# B&R Automation Studio project NAINV104C00R8L515F00 (part 2)

### Update LogProgram.txt
```
2023_08-10(R8)
Add LCSLF Phase2

Add Display of the Languages and Time
	UI	- Act_Background - P1000_ LangTime - Update the arrangement and display of the Languages and time
	NtParam - Add Chinese & German Prep

Manual Accept Condition Modification
	1)	LFFollower, Follower1, Follower2, etc.:
 		> Act_Background_AccData Script
	2) LCSLF:
	    > Act_Main Script
	3) USHermes:
    	> Act_Background_AccData Script
	UI:
	4) Act_OptP0200ToP0201AccDat

After power cycle the machine, buzzer will sound on due to the safety relay haven’t reset.

	DInput > Act_Background

Debug for Inshutter Hide in UI when Inlet Shutter disable in Ntparam.

2023-07-03(R7)
Add - Invert Once(PassThrough > Return & Invert) and Invert Twice(Invert > Return & Invert) Mode with Clmap(NoStopper)

	UI		> P0200 - add Upstream 2 Indication,PCB Reset
			> P1023 - add Upstream Selection
			> P0940	- Communication Control

	SMEMA	> Add - USSMEMA 2

	Conv	> Add - Conveyor Direction Access in Act_Link

	Operations	> Add - Act_OpsClampNoStopperInvOnceAndTwice, Act_Link

	McParam	> USCom2 Mod,Param,Selection
	NtParam > InvertOnce Prep, InvertTwicePrep, USSMEMA2Prep, RetrnBrdConvDir
	DI/DO	> Upstream SMEMA2
	Alarm 	> Latest Version

2023-05-08
Ops,ActLink p_bGoToStandby linked to USAllow

2022-08-12

DInput - Act_background, add Safety Relay Reset Alarm
FTP - Add addition user to access FTP

2022-04-01
ProdRcp -Act_Main,Act_EntP1040Disp,Act_OptP1040Save,Act_OptP1040Del,Act_OptP1040ToXML,Act_OptP1040FromXML,Act_EntP0400Disp

2022-06-10 (R5)
Hermes - Act_Link - Add flippedboard feature

2022-05-04
LFFollower, Follower1, DInput - Act_Link -  Add another US width check sensor at remote side.

2021-12-29
LFFollower, Follower1 - Act_Background - Add p_bDBAOnWOAllign to fbFolllower to send DBA even width check sensor is not alligned.

2021-10-19
CANOpenServo - Act_Background - Add error code for Estun Servo Motor.
                              - Reset control word 6040.4 to 0 when servo motor is in position

2021-09-01
LFLeader, LFFollower - Local,Input_Ref variables - Modify Product Recipe Related Variables to STRING[254]
LFFollower - Act_Background - Modify bUSAllow To Include p_bInternalReqProdRcpDiff

2021-06-19
R4 - Debug LF stopper extend retract bug

2021-06-12
R3 - P1021 - Debug Auto Log Out Time save problem.
   - Add Inverter_XStd_WShutter & Inverter_XStd_WClamp in Configuration View

2021-05-18
LFFollower - Act_Link - Change Info Message
		   - Act_Background, Act_Background_AccData - Change Product NameNot Exist and Width Mismatch Error To Info
		   - Act Main_Disable - Reset Variables When Function Is Disabled
Follower1  - Act_Background, Act_Background_AccData - Change Product NameNot Exist and Width Mismatch Error To Info
		   - Act Main_Disable - Reset Variables When Function Is Disabled

2021-04-20
Alarm - Act_Background - Add bInfoLF.
LFLeader - Act_Main - remove input for sequential mode (one time or always active)

2021-02-24
LFLeader - Act_Main - add input to select sequential mode (one time or always active)
LCS - Act_Link - Debug of second width parameter being empty when passing from LCS
2021-02-22
LifterBtm - Act_Link -> Add InterruptSensor3.

2021-02-18
Update - Visu - C0005
Update - UI - UI Folder - Act_Background - Act_OptC0005ChgPage.

2021-02-17
CANOpenServo - Act_Background - PosDiff updated from 50 to 500.
			 - Act_Alarm - udiCode change to 10299
			 - Local.var - update alarm message a_tyAlmText[10298] and a_tyAlmText[10299]

2021-01-11
TLBuz - Update Act_Background1, Act_Background2, Act_Background3.

2020-11-19
NtParam		 - Add variable bMagSafetyBarOrientation
Operations	 - OpsMagSafetyBar - ActOpsRun - Add p_bMagSafetyBarOrientation

2020-11-11
Tuning.diAsdaA2FirstTorqueCmd default setting is 300 in NtParam for all Delta servo motor.

2020-10-06
DOutput		 - Act_Link - add p_tyDISettings.diPCBOutJamSen > 0
			 - Act_InitGlobal - add p_tyDISettings ACCESS p_NtParamDISettings;
			 - Act_InitLocal - add p_tyDISettings ACCESS ADR(tyDISettings);

2020-10-05
Startup 	 - Act_Main_GetHWInfo - Debug Steps In Network Recovering
LFLeader 	 - Act_Initial, Act_Background_Process and Local.var - Rename and change the type of fbBlkUS to fbBlkUSDS
LFFollower, Follower1 - Act_Background, Act_Background_AccData - Add bLeaderOnline, replacing the direct usage of tyLeaderInfo.bOnline

2020-09-22
LFFollower 	 - Reset bLeaderSeqCtrlInActive in Act_Main_Disable.
HWInfo.typ 	 - Add One Enumeration (eNetworkConfigMod) & Two Actions (fbGetETHConfigMode and fbSetETHConfigMode) - Retrieve Or Set Network Configuration Of The PLC.
HWInfo 		 - Init, InitGlobal, InitLocal, Act Main, Act_Initial, Local.var and InputRef.var - Add The Additional Actions Related Variables
McParam  	 - McParam.typ Add eNetworkMod in tyMcParam.
NtParam  	 - NtParam.typ Add tyNetworkMOde (UILmt) in tyNtParam.
Startup	   	 - InitGlobal, InitLocal, Act_Main_GetHWInfo - Add Function To Load Saved Network Configuration s When New Configuration Detected.
		   	   InputRef_Link.var, InputRef.var & Local.var - Add New Startup Function Variables.

2020-09-16
McParam  	 - McParam.typ Add sIPAddr & sSubnetMask in tyMcParam.
HWInfo	 	 - Init, InitGlobal, InitLocal, Act_Main_GetHWInfo 	- Add Function To Load Saved IP Parameters When New IP Detected.
		   	   InputRef_Link.var, InputRef.var & Local.var 	- Add New HWInfo Function Variables.

2020-09-10
DSHermes 	 - Init, Cyclic, Act_Background_TCPListen, Act_Alarm4 - Improvise Alarm For Connection Lost.
		   	   Local.var - Add New Alarm Variables & Modify Alarm Text.

2020-08-24
LiftMagConv  - Act_Link - add fbSenOn1 for left sensor	by aiman
TopMagConv 	 - Act_Link - add fbSenOn2 for left sensor	by aiman
OpsMagLdr 	 - Act_OpsRun - changed condition in MagConvStepMagConv for Mag Exit

2020-08-17
LibVer 		 - Act_Main - Modify Function To Function Block In LibVerActReadChk.
		 	   Act_Initial - Initialize Newly Added Function Blocks.
		 	   Local.var - Declare New Function Blocks.

2020-08-06
NtParam.typ  - Add Two Actions (NtParamSave and NtParamLoad) - Export and import NtParam in XML Format
NtParam Act Main, Act_Initial, tyNtParam, InitLocal, Local.var and InputRef.var - Add The Additional Actions Related Variables
TLBuz 		 - All Act_Backgrounds Change Manual Mode Towerlight To Cater For Error Indication
LFLeader 	 - Add More Tags For Improving Leader Follower Concept, Modify p_diReqProdWidth To Use Downstream Width
LFFollower,
Follower 1 	 - Add fbOnlineChk For Leader Online Status
			 - Modify Act_Initial,Act_Background, Act_Background_AccData
			 - Add eCurrMachineStat For Status Indication
ProdRcp.typ	 - Add second width
LibVer 		 - Act_Main - Modify LibVerActReadChk, Add Step To Check File Validity.
		 	   Local.var - Add Alarm Text For File Coruption.

2020-07-24
MagRcp 		 - Add One Action in Act Main - MagRcpActSort
ProdRcp,	 - p_sSearch and sSearch in Local changed to STRING[254]
MagRcp 		 - sRcpNm for RcpParam in both ProdRcp.typ and MagRcp.typ temporary changed to STRING[30]

2020-06-30
Revert Traverser Main.st and AWClose Background.st program.
Add Estun error code "65362: sAxisErrTxt := 'Torque output alarm'";

2020-06-08
ProdRcp 	 - Increase Product Recipe Name Length to 254, Add Two Actions in Act Main - ProdRcpActSort & ProdRcpActEndCharFilter
LibVer 		 - Act_Main - LibVerActReadChk, made error if library data files corrupted.

2020-06-05
MagConv 	 - Update the Status of Mag Conv.Add one Action - MagConvActEntToMid.

2020-06-01
Stepper 	 - New package for stepper control.
MotorBrk 	 - Renewed package. Added MotorBrkActSetMtrDirOrCCW1 and MotorBrkActRstMtrDirOrCCW1.
	 	 	 - Modified fbRotCW and fbRotCCW and the access type to fbConvSenToSenBrkTm2Lmt.
	 	 	 - Added diMtrSigOnDlyTm (500), diMtrDirOffDlyTm (500), diMtrBrkOnDlyTm(100).

2020-04-28
MagConv 	 - Add MagConvActEntToMid Action.

2020-03-20
NtParam  	 - Add the selection of Motor model.

2020-03-16
TLBuz 		 - Add two inputs for buzzer behaviour, towerlight flash function to act_background and reset fbwarning.

2019-12-24
LFLeader 	 - Remove fbBlkDS2 in Act_Initial & Act_Background_Process, add pa_bLFOnline in Act_Background_Process

2019-10-31
TLBuz 		 - Regroup Structure Into Nutek, Aptiv & MEK.
MagConv 	 - Separate Program Into MagConv1Clamper & MagConv2Clamper.

2019-10-21
MagConv 	 - Improve with Action MagConvActPreExit & MagConvActPreExitClpr.
LFFollower 	 - Improve Change All Function Without Manually Accept Data.
LFLeader 	 - Add Second Oven Index, Improve Change All Function Without Manually Accept Data.
OpcUaMap.uad - Enable bBypassMnlAccDat Tag Name.
Startup 	 - Act_Main_SDOWrite, Remove SDOWrite.
CANOpenServo - Change Structure Of SDOWrite And Abnormal Movement.

2019-07-30
CANOpenServo - Due To Upgrade of NtMotion.

2019-07-18
LFFollower 	 - Act_Link, Minor debug.

2019-07-15
LCS 		 - Act_Link, Check Recipe Name Must Not Exceed 15 Char.

2019-07-10
LCS 		 - Add More Parameter For Live Data.

2019-07-04
LFFollower 	 - Improve of Recipe Compare Method For p_tyInternalReqProdRcp, tyUpdtProdRcp & tyRlsBrdProdRcpNm.

2019-07-03
LFFollower 	 - Improve Act_Background To Check Whole Product Recipe Different Instead of Name & Width Only.
Buffer 		 - Add p_tyBufferStat & p_tyDispBuffer And Improve For Two Program Control One Memory.

2019-06-28
USHermes 	 - Improve of Act_Background_AccData.
DSHermes 	 - Move of Act_Background_ChgConfig.
Buffer 		 - Improve of bParamDiff Condition.
LCSLF 		 - Improve of LCSActRunProd.

2019-06-27
LFFollower 	 - Improvement To Change Name & Width To Whole Product Recipe Type.

2019-06-17
Conv 		 - Add Two Action : ConvActEntToInOff & ConvActRevImmedStart.

2019-06-12
LFFollower 	 - Add Act_Background_ChkRlsBrd. Improvement of Act_Background_UpdtData.
LCSLF 		 - Add Update Data in Act_Background.

2019-06-11
TLBuz 	 	 - Modify ChgRcp.
LFFollower 	 - Improvement of UpdtData.

2019-06-10
ProdRcp 	 - Update tyCurrRcp To a_tyCurrRcp (Array).
LFFollower 	 - Add p_bInternalUse.
USHermes 	 - Add p_bInternalUse.
DSHermes 	 - Add p_bInternalUse.

2019-06-07
TLBuz 		 - Add Warning & ChgRcp.
TCP 		 - Add Start Code & End Code Checking.
Buffer 		 - Improve bParamDiff. Add bFIFOOld.

2019-06-04
USHermes 	 - Improvement At Accept Date (Act_Background_AccData).

2019-06-02
TCP 		 - New.

2019-05-30
Hermes 		 - Debug CheckAlive. SequenceTO Start Only After Connection Establish.
Flatstream 	 - Debug Act_Main.
USHermes 	 - Update Act_Link to Accept New Recipe.

2019-05-29
DVFrame 	 - Change From RS232. Improvement & Debug.
Flatstream 	 - New.

2019-05-28
MagConv 	 - Add MagConvActInitClpStop.
DCConv 		 - Improvement of DC Motor Alarm Trigger Time.
LFFollower 	 - Improve of Act_Background.
LCS 		 - Add "Warning" & "Info" For Live Data.

2019-05-27
LFFollower 	 - Debug Act_Link.
LCS 		 - Debug Act_Link. Add sErrMsg.
Buffer 		 - Debug Act_Main_Bffr. Add bMagRemoved.
Data 		 - Update of Default User.dat.

2019-05-24
LFFollower 	 - Improve of Act_Background.
MagConv 	 - Add MagConvActEntClpStop.
TLBuz 		 - Modify Warning Condition.

2019-05-22
OpcUaMap.uad - Update Tag Name.
LF 			 - Modify Set Time. Improve Of Act_Background for Accept Data.
LFLeader 	 - Add New Tag Name.
Time 		 - Update of Act_InitGlobal For LF Sync Time.
LCS 		 - Update To Reset If Receive Idle From LCS.

2019-05-21
RS232 		 - Add FullReadUntilValid.
LCS 		 - Move Some Program From Act_Background To Act_Link. Bug Fixed.

2019-05-20
RS232 		 - Modify to work with start code & end code.
ProdRcp 	 - Modify on dtLastModified in Act_LinkAction.
LCS 		 - Act_Background Show Boolean & dtLastModified Working Sample. Add Function Enable.
TLBuz 		 - Add Aptiv Mode.

2019-05-18
Buffer 		 - Check Next Unload Ignore Product Name.

2019-05-15
OvenInfo 	 - Improve of Act_Background.
Buffer 		 - Add bParamDiff to check current parameter and request parameter different.

2019-05-14
LCS 		 - Update Act_InitGlobal.
RS232 		 - New.

2019-05-11
LFFollower 	 - Improve And Able To Ignore MagRcp If Necessary.

2019-05-10
TLBuz 		 - Add Simulation Mode.
ProdRcp 	 - Improve Act_LinkAction.
Buffer 		 - Improve Act_LinkAction.
HWInfo 		 - Improve Act_Main While In Simulation.

2019-05-09
CANOpenServo - Improve of Error Axis Move Abnormally By External Force (10000).
ProdRcp 	 - Debug Write Recipe. Add Save List.
MagRcp 	 	 - Debug Write Recipe. Add Save List.
UsrFolder 	 - Create LCS Directory.
Startup 	 - Act_Main_UsrFolder, Create LCS Directory.
Alarm 		 - Combine Two Alarm Info.

2019-05-08
RmtHermes 	 - Debug Log title.
UsrMgmt 	 - Add Access Right Output.

2019-05-07
MagConv 	 - Debug.
ConvBffr 	 - Add Individual Have Board Output.
LF 			 - Major update.
LCSLF 		 - Change Name to tyCurrProdRcp.
ProdRcp 	 - Add Write Recipe Parameter.
MagRcp 		 - Add Write Recipe Parameter.
LCS 		 - Update to match LCS (PC).

2019-05-04
MagRcp 		 - Split Current Magazine Recipe From McParam.
ProdRcp 	 - Split Current Product Recipe From McParam.
UsrMgmt 	 - Split Access Right From McParam. Remove Nutek User.
Hermes 		 - Split Configuration From McParam. Add RmtHermes.
Startup 	 - Split Parameters From McParam. Add RmtHermes.
Remove "File Device" "NutekUser". Please Refer Configuration "4PPC30_043F_21F001".

2019-05-01
Hermes 		 - Log file change to day instead of hour. Due to startup too long to check old log when production run for long.

2019-04-30
LCS 		 - Improve To Match LCS (PC).
LFLeader 	 - Make a_tyFollowerToLeaderTag as Output.
All 		 - sStatTxt & a_sStatText Change To String[200].
ProdRcp 	 - Modify For LCS.

2019-04-28
MpProdRcp 	 - New.
Add "Config.mprecipexml" Under Configuration View > mapp. Please Refer Configuration "4PPC30_043F_21F001".
Add "File devices" For "MpProdRcp". Please Refer Configuration "4PPC30_043F_21F001".
Startup 	 - Modify Due To MpProdRcp.

2019-04-27
DSSMEMA 	 - Update due to NtSMEMA upgrade.

2019-04-26
Buffer 		 - Debug tyBuffer to p_tyBuffer. Improve bLastProductUnload Condition In Unload Board.
Startup 	 - Get Retain ConvBffr.
ConvBffr 	 - Update Link with Startup. Improve bLastProduct Condition In Remove Board. Add Have Board Output.
LFFollower 	 - Improve Act_LinkEn. Add Condition in Act_Link to update current recipe into leader tag.

2019-04-25
LibVer 		 - Modify To Move LibVer From "Private" To "User".
Update "File devices" For "LibVer". Please Refer Configuration "4PPC30_043F_21F001".
Add "File devices" For "LCS". Please Refer Configuration "4PPC30_043F_21F001".
Modify "FTP Server" "Users". Please Refer Configuration "4PPC30_043F_21F001".
Modify "OpcUaMap.uad". Please Refer Configuration "4PPC30_043F_21F001".
LFLeader 	 - Improvement.

2019-04-24
CANOpenServo - Add actual limit sensor output.
ProdRcp 	 - Add "Add" & "Edit" action. Improve of Act_LinkAction to suit LCS.
LCS 	 	 - New.

2019-04-23
LFLeader 	 - New.

2019-04-21
USHermes 	 - Modify Alarm Info.
LFFollower 	 - New.

2019-04-18
ConvBffr 	 - New.
Buffer 		 - Change of NtBffr.

2019-04-17
CANOpenServo - Remove Extra Homing Parameter, All Use Under tyMotionCANParamInHm.

2019-04-16
Operations 	 - Remove Accept Data & New Data.
Hermes 		 - Debug Log File. Modify Accept Data.

2019-04-11
USHermes 	 - Debug Log by adding step. Add p_bAccDataRdy.
DSHermes 	 - Debug Log by adding step.

2019-04-10
Startup 	 - bNtSettingsLoadDone should be FALSE as default.

2019-04-09
Ops2 		 - Update of p_bAccDat interlock by Ops1.
USHermes 	 - Update AccDatStep in Act_Link. Remove p_bChkBrdAvl. eStatus2 = Error then bRdyRcv = false. Update Act_Background_BoardAvailableChk. Add Manual Accept Data.
DSHermes 	 - Make local.var BoardAvailable new board parameter to default value.
NtParam 	 - Change of Act_LinkAction.
TLBuz 		 - Change of Act_LinkAction.
Buffer 		 - Change of Act_LinkAction.
Conv 		 - Change of Act_LinkAction.
DCConv 		 - Change of Act_LinkAction.
MagConv 	 - Change of Act_LinkAction.
MotorBrk 	 - Change of Act_LinkAction.
ConvSpd 	 - Change of Act_LinkAction.
SMEMA 	 	 - Change of Act_LinkAction.
Pneu 		 - Change of Act_LinkAction.
CANOpenServo - Change of Act_LinkAction.
Hermes 		 - Change of Act_LinkAction.

2019-04-08
DSHermes 	 - Minor debug on fbParseBrdAvlExternal.
Hermes 		 - Add program Hermes for board available memory use.
Startup 	 - Due to change of Hermes.

2019-04-04
OvenInfo 	 - Add p_bBGRun.
Startup 	 - Change eStartupStep member order for better display in UI.
UsrMgmt 	 - Add UsrMgmtActUsrBypassLogin & UsrMgmtActNtBypassLogin.
DSHermes 	 - Debug BoardAvailable for "New" and "External".
UI 			 - Remove Not Use Page.

2019-03-29
All 		 - Add Act_LinkAction.

2019-03-28
Startup 	 - Change "DelOldLogFile" to "Alarm". Add "Hermes". Error will reset Action to IDLE.

2019-03-25
All 	 	 - Change Action become input. Merge Alarm Text & Recovery Text into one type.

2019-03-22
Startup 	 - Add bNtSettingsLoadDone. Move StartupStepParameter after StartupStepUsrFolder in Act_Main.st.
All 		 - Update to match latest method of NtParam.

2019-03-16
Startup 	 - Act_Main_Bffr. Add BufferActBGStartCoolFan in Step 8.

2019-03-15
Hermes 		 - New Release

2019-03-13
UsrFolder 	 - Debug of Log directory path. Add "FileDevice" for "Log".

2019-03-11
DCConv 		 - Minor debug.

2019-02-26
AWClose 	 - Minor debug.

2019-02-23
Alarm 		 - Minor debug.
UsrFolder 	 - Add Create Log Directory.
Startup 	 - Improve of "Act_Main_UsrFolder" due to UsrFolder update.

2019-02-22
CANOpenServo - Change of Act_Action.

2019-02-21
DOutput 	 - Add Act_Link.

2019-02-20
DCConv 		 - Debug of ConvEngage.
CANOpenServo - fbModuleOK delay time change to 5s.

2019-02-19
CANOpenServo - Reset Error need to reset control word 6040.
TLBuz 		 - Improve of condition while p_bManual = True.

2019-02-18
Buffer 		 - Add background control of cool fan run.

2019-02-15
Conv 		 - Improve of condition while p_bManual = True.
DCConv 		 - Improve of condition while p_bManual = True.
MagConv 	 - Improve of condition while p_bManual = True.
MotorBrk 	 - Improve of condition while p_bManual = True.
SMEMA 		 - Improve of condition while p_bManual = True.

2019-02-14
ConvSpd 	 - Improve of condition while p_bManual = TRUE.
Change of Cyclic Time.
CANOpenServo - Change of Position Different Threshold.
Convert Library Into Binary

2019-02-11
TLBuz 		 - Warning Rest Time Change To 5s.
Buffer 		 - Add Magazine Present Timer.

2019-01-27
Buffer 		 - Add error code.

2019-01-26
Buffer 		 - Debug.

2019-01-25
Buffer 		 - Debug a_bSkip array size.
Lifter 		 - Debug Act_Background.
User.dat & NtUser.dat update.

2019-01-24
Pneu 		 - Modify Cyclic for disable.
AW 		 	 - Add GoWidthOff to turn off motor after auto width move.
Lifter 		 - Debug.
Traverser 	 - Debug.
Buffer 		 - Debug. Add background update display.
OvenInfo 	 - Modify Act_Main_Disable.

2019-01-23
Lifter 		 - Major debug in slot calculation. Add FullMovRel.
CANOpenServo - Debug reset error. Debug Act_Alarm.
DCConv 		 - Debug reset error.
Machine 	 - Debug reset error.
Operation 	 - Debug reset error.

2019-01-22
CANOpenServo - Minor debug.

2019-01-21
DInput 		 - Debug reset error.
CANOpenServo - Add eMainStatus. Add bJogging.
Time 		 - Add eMainStatus.
Operations 	 - Rename eStatus & udiStatus.

2019-01-20
Operations 	 - Update Structure.
SMEMA 		 - Update due to Library update.
Buffer 		 - Add error code.

2019-01-19
TLBuz 		 - Add Warning.

2019-01-18
RstErr 		 - Act_Main update.
CANOpenServo - Add output. Set Default Value for siModOfOptDisp_6061:=6.
Change of Cyclic time.
Buffer 		 - Update Local.var
Add file for NtUser, LibrariesVersion & User.
Conv 		 - Add Pneu status output.
DCConv 		 - Add Pneu status output.
Operations 	 - Modify structure in Cyclic.

2019-01-17
DCConv 		 - Act_Main debug.

2019-01-16
Trav 		 - Remove diPitch.
Lifter 		 - Remove diPitch.
Operations 	 - Modify Reset methos.

2019-01-15
McParam 	 - File name as input.
NtParam 	 - File name as input.
Buffer 		 - File name as input.
Operations 	 - Add bAccData.

2019-01-14
Operations 	 - Update Alarm & Sequence.
SMEMA 		 - bTimer & bVirtual as output. Debug Act_Background timer interlock.

2019-01-12
Conv 		 - Convert time out type.
DCConv 		 - Convert time out type.
MagConv 	 - Convert time out type.
OvenInfo 	 - diBrdInOven change to retain.
SMEMA 		 - Update timer condition. Add bComplSigOn.
Startup 	 - Debug for HWInfo.

2019-01-11
SMEMA 		 - Minor debug. Add Act_LinkEn.
Operations 	 - Add alarm. Add Act_LinkEn.
MagRcp 		 - Add Act_LinkEn.
OvenInfo 	 - Add Act_LinkEn. Minor debug.
Conv 		 - Add Act_LinkEn. Add conveyor time out.
DCConv 		 - Add Act_LinkEn. Add conveyor time out.
MagConv 	 - Add Act_LinkEn. Add conveyor time out.
MotorBrk 	 - Add Act_LinkEn.
ConvSpd 	 - Add Act_LinkEn.
RS232Mirtec  - Add Act_LinkEn.
Pneu 		 - Add Act_LinkEn.
CANOpenServo - Add Act_LinkEn. Major Update.

2019-01-10
McParam 	 - Remove ProdRcpWrite & MagRcpWrite.
OvenInfo 	 - Act_Main modify for change of eStat.
Conv 	 	 - Act_Main modify for change of eStat.
DCConv 		 - Act_Main modify for change of eStat.
MagConv 	 - Act_Main modify for change of eStat.
MotorBrk 	 - Act_Main modify for change of eStat.
ConvSpd 	 - Act_Main modify for change of eStat.
SMEMA 		 - Act_Main modify for change of eStat.
DOutput 	 - Act_Main modify for change of eStat.
Pneu 		 - Act_Main modify for change of eStat.
Operations 	 - Act_Main modify for change of eStat.

2019-01-09
AW 			 - Update bWidthPosDiff when disable.
Lifter 		 - Update bSltPosDiff when disable.
Conv 		 - Add bGdBrdInit. Debug tMtrOffDlyTm. Improve Act_Action to let eStatus = DONE also able change eStat directly.
DCConv 		 - Add bGdBrdInit. Improve Act_Action to let eStatus = DONE also able change eStat directly.
SMEMA 		 - Add tRstDlyTm. Improve Act_Action to let eStatus = DONE also able change eStat directly.
Operations 	 - Add Act_Main_Disable. Improve Act_Action to let eStatus = DONE also able change eStat directly.
TLBuz 		 - Improve Act_Action to let eStatus = DONE also able change eStat directly.
OvenInfo 	 - Improve Act_Action to let eStatus = DONE also able change eStat directly.
MagConv 	 - Improve Act_Action to let eStatus = DONE also able change eStat directly.
MotorBrk 	 - Improve Act_Action to let eStatus = DONE also able change eStat directly.
ConvSpd 	 - Improve Act_Action to let eStatus = DONE also able change eStat directly.
DOutput 	 - Improve Act_Action to let eStatus = DONE also able change eStat directly.
Pneu 		 - Improve Act_Action to let eStatus = DONE also able change eStat directly.

2019-01-08 //Until Here////
DOutput 	 - Add output.
SMEMA 		 - bTimer will be trigger only during SMEMAActRun.
Operations 	 - Combine Ops1 & Ops2 into Ops.

2019-01-07
SMEMA 		 - Add bUSRdy, bUSGdBrdRdy & bDSRdy for USSMEMA & DSSMEMA.
Conv 		 - Add tMtrOffDlyTm.
DCConv 		 - Add tMtrOffDlyTm.
MagConv 	 - Add tMtrOffDlyTm.
Time 		 - Combine Error
CANOpenServo - Combine Error
Alarm 		 - Remove link data.

2019-01-04
Machine 	 - Debug Act_Alarm1.
Time 		 - Debug Init.st.
Operations 	 - Debug Ops1 > Act_Main. Add sStepTxt into Act_Main. Add Act_Dummy.
Conv 		 - Due to NtConv update, add one more type of Exit.
DCConv 		 - Due to NtConv update, add one more type of Exit.
MagConv 	 - Due to NtConv update, add one more type of Exit.
SMEMA 		 - Add Timer & Virtual.

2019-01-03
Machine 	 - Debug Act_Alarm & Act_Alarm1. Modify background error handling.
CANOpenServo - Modify background error handling. Update sStatTxt in Act_Initial.
AW 			 - Replace diStandPitchInUM (Input) to diPitchInUM (Local).
Time 		 - Modify background error handling. Update sStatTxt in Act_Initial.
DCConv 		 - Modify background error handling. Update sStatTxt in Act_Initial.
DInput 		 - Modify background error handling.
UsrMgmt 	 - Update sStatTxt in Act_Initial.
McParam 	 - Update sStatTxt in Act_Initial.
NtParam 	 - Update sStatTxt in Act_Initial.
ProdRcp 	 - Update sStatTxt in Act_Initial.
MagRcp 		 - Update sStatTxt in Act_Initial.
HWInfo 		 - Update sStatTxt in Act_Initial.
UsrFolder 	 - Update sStatTxt in Act_Initial.
LibVer 		 - Update sStatTxt in Act_Initial.
General 	 - Update sStatTxt in Act_Initial.
TLBuz 		 - Update sStatTxt in Act_Initial.
OvenInfo 	 - Update sStatTxt in Act_Initial.
Buffer 		 - Update sStatTxt in Act_Initial.
RstErr 		 - Update sStatTxt in Act_Initial.
Conv 		 - Update sStatTxt in Act_Initial.
MagConv 	 - Update sStatTxt in Act_Initial.
MotorBrk 	 - Update sStatTxt in Act_Initial.
ConvSpd 	 - Update sStatTxt in Act_Initial.
Alarm 		 - Update sStatTxt in Act_Initial.
RS232Mirtec  - Update sStatTxt in Act_Initial.
SMEMA 		 - Update sStatTxt in Act_Initial.
UI 			 - Update sStatTxt in Act_Initial.
DOutput 	 - Update sStatTxt in Act_Initial.
Pneu 		 - Update sStatTxt in Act_Initial.
Operations   - Update sStatTxt in Act_Initial.
Startup 	 - Update sStatTxt in Act_Initial.

2019-01-02
UsrMgmt 	 - Change of sStatTxt update.
McParam 	 - Change of sStatTxt update.
NtParam 	 - Change of sStatTxt update.
ProdRcp 	 - Change of sStatTxt update.
MagRcp 		 - Change of sStatTxt update.
Time 		 - Change of sStatTxt update.
HWInfo 		 - Change of sStatTxt update.
UsrFolder 	 - Change of sStatTxt update.
LibVer 		 - Change of sStatTxt update.
General 	 - Change of sStatTxt update.
TLBuz 		 - Change of sStatTxt update.
OvenInfo 	 - Change of sStatTxt update.
Buffer 		 - Change of sStatTxt update.
RstErr 		 - Change of sStatTxt update.
Conv 		 - Change of sStatTxt update.
DCConv 		 - Change of sStatTxt update.
MagConv 	 - Change of sStatTxt update.
MotorBrk 	 - Change of sStatTxt update.
ConvSpd 	 - Change of sStatTxt update.
Alarm 		 - Change of sStatTxt update.
RS232Mirtec  - Change of sStatTxt update.
SMEMA 		 - Change of sStatTxt update.
UI 			 - Change of sStatTxt update.
DOutput 	 - Change of sStatTxt update.
Pneu 		 - Change of sStatTxt update.
Operations 	 - Change of sStatTxt update.
CANOpenServo - Change of sStatTxt update. Update eStatus to Busy while running.
Startup 	 - Change of sStatTxt update.

2018-12-31
CANOpenServo - Seperate input reference.

2018-12-27
Time 		 - Remove bBGRun.
TLBuz 		 - Remove bBGRun. Add manual reset.
OvenInfo 	 - Background direct link to input bPrepExtdd, bEnExtdd & bDisExtdd. Add manual reset.
Buffer 		 - Background Cool Fan Control direct link to input bPrepCoolTm & bCoolFanTm.
DCConv 	 	 - Remove bBGRun. Add manual reset.
AlarmLog 	 - Background run is control by Action.
Machine 	 - Remove bBGRun.
SMEMA 		 - Remove bBGRun. Add manual reset.
DInput 		 - Remove bBGRun.
DOutput 	 - Remove bBGRun. Add manual reset.
CANOpenServo - Remove bBGRun. Background run is control by Action. Add manual reset.
AW 			 - Add bWidthPosDiff.
Lifter 		 - Add bSltPosDiff.
Startup 	 - Background run is control by Action. Shorten local variable name.
McParam 	 - Add McParam program without Magazine (McParam2).
RstErr 		 - Add manual reset.
Conv 		 - Add manual reset.
MagConv 	 - Add manual reset.
MotorBrk 	 - Add manual reset.
ConvSpd 	 - Add manual reset.
Pneu 		 - Add manual reset.

2018-12-26
CPU 		 - Update distribute of program in CPU. Update cyclic time.
FTP 		 - Update of FTP server configurations.
Startup 	 - Remove bStartupErr.
HWInfo 		 - After set new IPAddr & Subnetmask will update output.
TLBuz 		 - Rising of bManual will set Amber Light ON.
Conv 		 - Remove functions reset in individual eStat.
MagConv 	 - Remove functions reset in individual eStat.
MotorBrk 	 - Remove functions reset in individual eStat.
DCConv 		 - New program.
Operations 	 - Update of OperationsActStep.

2018-12-24
Operations 	 - Add bRun.Sequence will execute base on bRun instead of bStatusRun.

2018-12-21
Buffer 		 - Add individual cooling fan control.
McParam 	 - Move Hermes parameter to Hermes program type.
MagConv 	 - Add bClprTwoOutputControl. Remove bClprUnclampCtrl.

2018-12-20
TLBuz 		 - Add bMuteBuz.
OvenInfo 	 - Add bDis.
Conv 		 - Add bEn.
MagConv 	 - Add bEn.
MotorBrk 	 - Add bEn.
ConvSpd 	 - Add bEn.
RS232Mirtec  - Add bEn.
SMEMA 		 - Add bDis.
Pneu 		 - Add bEn.
CANOpenServo - Add bEn.
CANOpenServo - AutoWidth - Add diMaxWidthInUM, diMinWidthInUM, diWidthOffsetInUM & diStdPitch.
Operations 	 - Add bPrep, bEn & bDis. Add OperationsStatusCycleStopping. Default Status is OperationsStatusStop. Add Boolean output for Status.
MagRcp 	 	 - Change sDisplayInfo & Magazine Parameter.
Startup 	 - Add bRun.

2018-12-14
RstErr 		 - Add bManual to control reset of output in Idle. Reset output in Idle after ManualMode off.
Conv 		 - Add bManual to control reset of output in Idle. Rename eAction. Reset output in Idle after ManualMode off.
ConvSpd 	 - Add bManual to control reset of output in Idle. Reset output in Idle after ManualMode off.
MtrBrk 		 - Add bManual to control reset of output in Idle. Rename eAction. Reset output in Idle after ManualMode off. Reset after change eStat.
MagConv 	 - Add bManual to control reset of output in Idle. Rename eAction. Reset output in Idle after ManualMode off. Reset after change eStat.
OvenInfo 	 - Set bOvenAllow to TRUE, if all functions not activated.
SMEMA 		 - Reset output in Idle after ManualMode off.
Pneu 		 - Add Extended & Retracted output.

2018-12-13
Conv 		 - Change of Conv2Sen to Conv. Add Reject & Inspection functions. Add individual output control.
Pneu 		 - Add bTwoCtrlIn & bTwoCtrlOut.
TLBuz 		 - Add individual output control.
ConvSpd 	 - Add individual output control.
OvenInfo 	 - Add individual output control. Move functions into Act_Background.
RstErr 		 - Add individual output control.
MtrBrk 		 - Add individual output control.
MagConv 	 - Add individual output control.
DOutput 	 - Add individual output control.
SMEMA 		 - Add individual output control.

2018-12-12
Startup 	 - Add Logout during User Management Startup.
Time 	 	 - Move Act_Background above Act_Main.
Buffer 		 - Move Act_Background above Act_Main.
Alarm 		 - Move Act_Background above Act_Main.
CANOpenServo - Move Act_Background above Act_Main.
Operations 	 - Change of Conv2Sen to Conv.

2018-12-11
DOutput 	 - Split to Act_InitGlobal & Act_InitLocal.
Pneu 		 - Change in all program. Add Pneu3Sen program.
Operations 	 - Update sample to 2 operations. Rename variable.
CANOpenServo - Rename variable.
```

### Update LogLibrary.txt
```
2022-07-05
NtRecipe 5.00.4 Debug of Sorting Function

2022-01-25
NtRecipe 5.00.4 - Improve fRecipeNmCompare

2021-12-29
NtLF 5.01.5 - Add bDBAOnWOAllign to send DBA even width check sensor is not alligned.

2021-10-19
NtMotion 5.00.9 - Uncheck servo on and homing operation if both have been done

2021-09-01
NtLF 5.01.4 - Modify Product Recipe Name Related Variables to STRING[254]

2021-04-20
NtLF 5.01.3 - Update fLFUSAllow & fLFDSAllow Block Conditions.
			- Modify fLFFollowerProdAccDataReq.

2021-02-24
NtLF:5.01.2 - Modify fLFUSAllow.

2021-02-23
NtSMEMA: 5.00.6 - Add fbSMEMATransporting1.

2021-02-17
NtMotion:5.00.8 - Limit sensor intelock for Estun Servo Movement. (20210217)
       - Homing timeout in 3 sec if home sensor broken.
       - Set default value for servo parameter if the NtParam setting out of the limit.

2020-11-10
NtMotion:5.00.7 - Torque limit setting at NtParam.

2020-10-05
NtLF:5.01.1 	 - Improve Change All For Section Leader, Debug Change Sequential.

2020-09-10
NtTCP:5.00.2 	 - Change of fbTCPClntConnect.

2020-08-17
NtVersion:5.01.1 - Change of fChkFileValidity & fInvalidCharInFileChk to function block.

2020-08-06
NtLF:5.01.0 	 - Improve leader follower concept.
				 - Add more tags in tyLeaderToFollowerTag and tyFollowerToLeaderTag.
NtVersion:5.01.0 - Add fChkFileValidity and fInvalidCharInFileChk.

2020-07-24
NtRecipe:5.00.3  - Debug of sorting functions.

2020-06-30
NtMotion:5.00.6  - Homing action when remote side limit sensor is on.

2020-06-15
NtMotion:5.00.5  - Homing timeout error when limit switch disconnected.

2020-06-08
NtRecipe:5.00.2  - Update Product Recipe to 254, Add Sorting and End Character Filter Functions.
NtVersion:5.00.1 - Debug of fChkLibrariesVer.

2020-06-07
NtUI:5.00.1 	 - Update fbTableCtrl and fbTableCtrl_v2. Update tyUILString.

2020-06-01
NtStepper:5.00.0 - New Release.
NtConv:5.00.3	 - Added fbConvSenToSenBrkTm2Lmt & fbConvSenToSenBrk2.

2020-03-20
NtMotion:5.00.4  - Add Estun Pronet, Schneider Electric Lexium 28 Servo Motor Control.
		 		 - Resolve Limit Switch Alarm when Delta servo motor perform homing at stratup of auto mode.

2020-03-16
NtTLBuz:5.00.2 	 - Add inputs to allow repeat sequence for fbTLBuzWarn.

2020-03-11
NtMotion:5.00.3  - Add Estun and Schneider.

2019-12-24
NtLF:5.00.5 	 - Modify fbLeaderBlkDS, include machine index before & after oven 2, block machine to machine when different width

2019-10-29
NtHermes:5.00.3  - Debug of fHermesGetTimeStamp

2019-10-21
NtRecipe:5.00.1  - Debug Of fRecipeGetInfo.
NtSMEMA:5.00.4 	 - fbSMEMAUS_9851, fbSMEMAUS_Std, fbSMEMADS_OppFirst, reset signal while error.
NtBuffer:5.00.6  - Debug of fBffrSetFull, fBffrSetMty for slot disable.
NtLF:5.00.5 	 - Add bBypassMnlAccDat Tag Name, Improve Change All Function Without Manually Accept Data.

2019-08-27
NtBuffer:5.00.5  - Debug of fBffrNxtLoadSeqAny, fBffrNxtLoadSeqGd & fBffrNxtLoadSeqBad.

2019-07-30
NtMotion:5.00.2  - Add Input To Select Homing Without Index Pulse.

2019-07-19
NtSMEMA:5.00.3 	 - fbSMEMADS, reset signal while error.

2019-07-03
NtBuffer:5.00.4  - Debug Of Limit Buffer Range.

2019-06-07
NtTLBuz:5.00.1 	 - Improve of fbTLBuzWarn.

2019-05-30
NtSMEMA:5.00.2 	 - Improve fbSMEMATransportIdle.

2019-05-29
NtRS232:5.00.2 	 - Add Flatstream Function.

2019-05-28
NtBuffer:5.00.3  - Debug of fBffrNxtLoadNearby.

2019-05-22
NtLF:5.00.3 	 - ChgAll Will Bypass Width Check Sensor.

2019-05-21
NtRS232:5.00.1 	 - Add fbFullReadUntilValid.

2019-05-17
NtMessage:5.00.1 - Debug When Attribute Value Is Empty String.

2019-05-07
NtConv:5.00.2 	 - After Time Out, Reset Output.
NtLF:5.00.2 	 - Debug fLFUSAllow. Modify fbLFFollower.

2019-05-04
NtHermes:5.00.2  - Debug Due to RmtHermes.

2019-04-27
NtSMEMA:5.00.1 	 - Improve Standard SMEMA According to Nutek Standard.

2019-04-25
NtHermes:5.00.1  - Debug fHermesIllegalMsgBrdAvlDS. To Handle MachineReady & StartTransport Send In One Message.

2019-04-23
NtLF:5.00.1 	 - Major upgrade.

2019-04-18
NtBffr:5.00.2 	 - Add Buffer Name, Product Name & Barcode.

2019-04-11
NtConv:5.00.1 	 - Debug of Time Out Error.

2019-04-04
NtBuffer:5.00.1  - Modify fBffrStat.

2019-04-02
NtTCP:5.00.1 	 - fbTPCSend & fbTCPRcv modify bEn = False condition. Disable check alive set function in Simulation Mode.

2019-03-25
NtGeneral:5.00.1 - Add tyAlmTxt.
NtLogFile:5.00.1 - Increase Alarm String Size.

2019-03-15
NtHermes:5.00.0  - New Release

2019-02-20
NtMotion:5.00.1  - Increase Module OK check counter from 5 to 20.
                 - Update fMotionModuleOK.
                 - Change of Position Different Threshold
// 5.00.0
2019-01-20
NtSMEMA 		 - Update.

2019-01-18
NtMotion 		 - Update for FwdLimit & RevLimit.

2019-01-11
NtSMEMA 		 - Update library.
NtConv 			 - Add time out.

2019-01-09
NtMotion 		 - Debug move absolute with backlash.

2019-01-08
NtMotion 		 - Debug move absolute with backlash.
NtConv 			 - Debug end sensor edgeneg trigger.

2019-01-04
NtConv 			 - Add fbConvSenToSenOff1.

2019-01-03
NtTCP 			 - Update.
NtMessage 		 - Update.
```

- User.dat (binary file, 3552 bytes)
- LibrariesVersion.dat (binary file, 2222 bytes)
### SoftwareVersion.var
```iecst
VAR CONSTANT
	sSWVersion : STRING[30] := 'NAINV104C00R8L515F00';
END_VAR
```

### Package Logical/Libraries - Global libraries

### Library Logical/NtLibraries/NtUI (IEC, version 5.00.2) - 5.00.2 - Add tyUIBitmap & tyUIBtn (uiValueIdx) to accomodate higher range of offset index (20210625)
5.00.1 - Update fbTableCtrl, fbTableCtrl_v2 and tyUILString.(20200608)
5.00.0 - New Library Design. (20181203)

#### NtUI.fun - Exported functions and function blocks
```iecst
FUNCTION fUIInRtStatOff : UINT (*Runtime Status Datapoint Off All Control*) (*$GROUP=Nutek,$CAT=User,$GROUPICON=Icon_Nutek.png,$CATICON=User.png*)
	VAR_INPUT
		uiRtStat : REFERENCE TO UINT; (*Runtime Status Datapoint*)
	END_VAR
END_FUNCTION

FUNCTION fUIInRtStatHide : UINT (*Runtime Status Datapoint Hide Control*) (*$GROUP=Nutek,$CAT=User,$GROUPICON=Icon_Nutek.png,$CATICON=User.png*)
	VAR_INPUT
		uiRtStat : REFERENCE TO UINT; (*Runtime Status Datapoint*)
	END_VAR
END_FUNCTION

FUNCTION fUIInRtStatLock : UINT (*Runtime Status Datapoint Lock Control*) (*$GROUP=Nutek,$CAT=User,$GROUPICON=Icon_Nutek.png,$CATICON=User.png*)
	VAR_INPUT
		uiRtStat : REFERENCE TO UINT; (*Runtime Status Datapoint*)
	END_VAR
END_FUNCTION

FUNCTION fUIInRtStatFocus : UINT (*Runtime Status Datapoint Focus Control*) (*$GROUP=Nutek,$CAT=User,$GROUPICON=Icon_Nutek.png,$CATICON=User.png*)
	VAR_INPUT
		uiRtStat : REFERENCE TO UINT; (*Runtime Status Datapoint*)
	END_VAR
END_FUNCTION

FUNCTION fUIInRtStatOpenTP : UINT (*Runtime Status Datapoint Open Touchpad Control*) (*$GROUP=Nutek,$CAT=User,$GROUPICON=Icon_Nutek.png,$CATICON=User.png*)
	VAR_INPUT
		uiRtStat : REFERENCE TO UINT; (*Runtime Status Datapoint*)
	END_VAR
END_FUNCTION

FUNCTION fUIOutRtStatCursor1Valid : BOOL (*Runtime Status Datapoint Cursor 1 Valid Output*) (*$GROUP=Nutek,$CAT=User,$GROUPICON=Icon_Nutek.png,$CATICON=User.png*)
	VAR_INPUT
		uiRtStat : REFERENCE TO UINT; (*Runtime Status Datapoint*)
	END_VAR
END_FUNCTION

FUNCTION fUIOutRtStatCursor2Valid : BOOL (*Runtime Status Datapoint Cursor 2 Valid Output*) (*$GROUP=Nutek,$CAT=User,$GROUPICON=Icon_Nutek.png,$CATICON=User.png*)
	VAR_INPUT
		uiRtStat : REFERENCE TO UINT; (*Runtime Status Datapoint*)
	END_VAR
END_FUNCTION

FUNCTION fUIOutRtStatTPIsOpen : BOOL (*Runtime Status Datapoint Touchpad Is Open Output*) (*$GROUP=Nutek,$CAT=User,$GROUPICON=Icon_Nutek.png,$CATICON=User.png*)
	VAR_INPUT
		uiRtStat : REFERENCE TO UINT; (*Runtime Status Datapoint*)
	END_VAR
END_FUNCTION

FUNCTION fUIOutRtStatOnLock : BOOL (*Runtime Status Datapoint Touch On Lock Output*) (*$GROUP=Nutek,$CAT=User,$GROUPICON=Icon_Nutek.png,$CATICON=User.png*)
	VAR_INPUT
		uiRtStat : REFERENCE TO UINT; (*Runtime Status Datapoint*)
	END_VAR
END_FUNCTION

FUNCTION fUIOutRtStatHasFocus : BOOL (*Runtime Status Datapoint Has Focus Output*) (*$GROUP=Nutek,$CAT=User,$GROUPICON=Icon_Nutek.png,$CATICON=User.png*)
	VAR_INPUT
		uiRtStat : REFERENCE TO UINT; (*Runtime Status Datapoint*)
	END_VAR
END_FUNCTION

FUNCTION fUIOutRtStatInEdit : BOOL (*Runtime Status Datapoint In Edit Output*) (*$GROUP=Nutek,$CAT=User,$GROUPICON=Icon_Nutek.png,$CATICON=User.png*)
	VAR_INPUT
		uiRtStat : REFERENCE TO UINT; (*Runtime Status Datapoint*)
	END_VAR
END_FUNCTION
(**)

FUNCTION_BLOCK fbTouchGetAction (*Get Touch Action Coordinate*) (*$GROUP=Nutek,$CAT=User,$GROUPICON=Icon_Nutek.png,$CATICON=User.png*)
	VAR_INPUT
		sVisuNm : STRING[80]; (*Visualization Object Name*)
	END_VAR
	VAR_OUTPUT
		bPressed : BOOL; (*Touch Pressed*)
		udiX : UDINT; (*X Coordinate*)
		udiY : UDINT; (*Y Coordinate*)
	END_VAR
	VAR
		tyInternal : tyTouchGetActionInternal; (*Local Variables*)
	END_VAR
END_FUNCTION_BLOCK

FUNCTION_BLOCK fbTouchFilter (*Filter Touch Action*) (*$GROUP=Nutek,$CAT=User,$GROUPICON=Icon_Nutek.png,$CATICON=User.png*)
	VAR_INPUT
		bPressedIn : BOOL; (*Touch Pressed*)
		udiXIn : UDINT; (*X Coordinate*)
		udiYIn : UDINT; (*Y Coordinate*)
	END_VAR
	VAR_OUTPUT
		bPressedOut : BOOL; (*Touch Pressed*)
		udiXOut : UDINT; (*X Coordinate*)
		udiYOut : UDINT; (*Y Coordinate*)
	END_VAR
	VAR
		tyInternal : tyTouchFilterInternal; (*Local Variables*)
	END_VAR
END_FUNCTION_BLOCK

FUNCTION_BLOCK fbTouchGetSlideDist (*Record Touch Action*) (*$GROUP=Nutek,$CAT=User,$GROUPICON=Icon_Nutek.png,$CATICON=User.png*)
	VAR_INPUT
		udiWorkAreaStartX : UDINT; (*Valid Area Start X*)
		udiWorkAreaStartY : UDINT; (*Valid Area Start Y*)
		udiWorkAreaEndX : UDINT; (*Valid Area End X*)
		udiWorkAreaEndY : UDINT; (*Valid Area End Y*)
		udiMinXDist : UDINT; (*Minimum X Real Time Distance*)
		udiMinYDist : UDINT; (*Minimum Y Real Time Distance*)
		bPressed : BOOL; (*Touch Pressed*)
		udiX : UDINT; (*X Coordinate*)
		udiY : UDINT; (*Y Coordinate*)
	END_VAR
	VAR_OUTPUT
		diXDist : DINT; (*X Real Time Distance*)
		diYDist : DINT; (*Y Real Time Distance*)
	END_VAR
	VAR
		tyInternal : tyTouchGetSlideDistInternal; (*Local Variables*)
	END_VAR
END_FUNCTION_BLOCK

FUNCTION_BLOCK fbTouchGetTap (*Get Double Tap*) (*$GROUP=Nutek,$CAT=User,$GROUPICON=Icon_Nutek.png,$CATICON=User.png*)
	VAR_INPUT
		udiWorkAreaStartX : UDINT; (*Valid Area Start X*)
		udiWorkAreaStartY : UDINT; (*Valid Area Start Y*)
		udiWorkAreaEndX : UDINT; (*Valid Area End X*)
		udiWorkAreaEndY : UDINT; (*Valid Area End Y*)
		udiMinSingleTapXDiff : UDINT := 20; (*Minimum Single Tap X Difference*)
		udiMinSingleTapYDiff : UDINT := 20; (*Minimum Single Tap Y Difference*)
		tMaxDoubleTapTm : TIME := T#900ms; (*Minimum Double Tap Time*)
		udiMinDoubleTapXDiff : UDINT := 20; (*Minimum Double Tap X Difference*)
		udiMinDoubleTapYDiff : UDINT := 20; (*Minimum Double Tap Y Difference*)
		bPressed : BOOL; (*Touch Pressed*)
		udiX : UDINT; (*X Coordinate*)
		udiY : UDINT; (*Y Coordinate*)
	END_VAR
	VAR_OUTPUT
		bSingleTap : BOOL; (*Single Tap Valid*)
		udiSingleTapX : UDINT; (*Single Tap X Coordinate*)
		udiSingleTapY : UDINT; (*Single Tap Y Coordinate*)
		bDoubleTap : BOOL; (*Double Tap Valid*)
		udiDoubleTapX : UDINT; (*Double Tap X Coordinate*)
		udiDoubleTapY : UDINT; (*Double Tap Y Coordinate*)
	END_VAR
	VAR
		tyInternal : tyTouchGetTapInternal; (*Local Variables*)
	END_VAR
END_FUNCTION_BLOCK

FUNCTION_BLOCK fbTableCtrl (*Table Control*) (*$GROUP=Nutek,$CAT=User,$GROUPICON=Icon_Nutek.png,$CATICON=User.png*)
	VAR_INPUT
		sVisuNm : STRING[80]; (*Visualization Object Name*)
		udiWorkAreaStartX : UDINT; (*Valid Area Start X*)
		udiWorkAreaStartY : UDINT; (*Valid Area Start Y*)
		udiWorkAreaEndX : UDINT; (*Valid Area End X*)
		udiWorkAreaEndY : UDINT; (*Valid Area End Y*)
		udiMinXDist : UDINT; (*Minimum X Real Time Distance*)
		udiMinYDist : UDINT; (*Minimum Y Real Time Distance*)
		uiSlideScale : UINT := 1; (*Slider Scale*)
		iTotalData : INT; (*Total Number of Data*)
		iTotalRow : INT; (*Total Number of Row*)
		bSelectedRowMnl : BOOL; (*Manual Selected Row*)
		uiSelectedRowMnl : UINT := 1; (*Manual Selected Row*)
		bTablePosPlus : BOOL; (*Plus Table Position*)
		bTablePosMinus : BOOL; (*Minus Table Position*)
	END_VAR
	VAR_OUTPUT
		bTableActive : BOOL; (*Table Active*)
		bSliderActive : BOOL; (*Slider Active*)
		uiSelectedRow : UINT := 1; (*Selected Row*)
	END_VAR
	VAR_IN_OUT
		uiSliderStatus : UINT; (*Slider Status*)
		a_tyUIHotspot : ARRAY[1..15] OF tyUIHotspot; (*Array of Hotspot on Table*)
		uiTablePos : UINT; (*Table Position*)
		iSliderPos : INT; (*Slider Position*)
	END_VAR
	VAR
		tyInternal : tyTableCtrlInternal := (fbSingleTapChkDlyTm:=(PT:=T#500ms),fbSliderOffTm:=(PT:=T#5s),fbTouchGetTap:=(udiMinSingleTapXDiff:=20,udiMinSingleTapYDiff:=20,tMaxDoubleTapTm:=T#900ms,udiMinDoubleTapXDiff:=20,udiMinDoubleTapYDiff:=20),iTablePos:=1,iTablePosTemp:=1); (*Local Variables*)
	END_VAR
END_FUNCTION_BLOCK

FUNCTION_BLOCK fbTableCtrl_v2 (*Table Control*) (*$GROUP=Nutek,$CAT=User,$GROUPICON=Icon_Nutek.png,$CATICON=User.png*)
	VAR_INPUT
		sVisuNm : STRING[80]; (*Visualization Object Name*)
		udiWorkAreaStartX : UDINT; (*Valid Area Start X*)
		udiWorkAreaStartY : UDINT; (*Valid Area Start Y*)
		udiWorkAreaEndX : UDINT; (*Valid Area End X*)
		udiWorkAreaEndY : UDINT; (*Valid Area End Y*)
		udiMinXDist : UDINT; (*Minimum X Real Time Distance*)
		udiMinYDist : UDINT; (*Minimum Y Real Time Distance*)
		uiSlideScale : UINT := 1; (*Slider Scale*)
		iTotalData : INT; (*Total Number of Data*)
		iTotalRow : INT; (*Total Number of Row*)
		bSelectedRowMnl : BOOL; (*Manual Selected Row*)
		uiSelectedRowMnl : UINT := 1; (*Manual Selected Row*)
		bTablePosPlus : BOOL; (*Plus Table Position*)
		bTablePosMinus : BOOL; (*Minus Table Position*)
		p_bTableActive : REFERENCE TO BOOL; (*Table Active*)
		p_bSliderActive : REFERENCE TO BOOL; (*Slider Active*)
		p_uiSelectedRow : REFERENCE TO UINT; (*Selected Row*)
		p_uiSliderStatus : REFERENCE TO UINT; (*Slider Status*)
		pa_tyUIHotspot : REFERENCE TO ARRAY[1..15] OF tyUIHotspot; (*Array of Hotspot on Table*)
		p_uiTablePos : REFERENCE TO UINT; (*Table Position*)
		p_iSliderPos : REFERENCE TO INT; (*Slider Position*)
	END_VAR
	VAR
		tyInternal : tyTableCtrlInternal := (fbSingleTapChkDlyTm:=(PT:=T#500ms),fbSliderOffTm:=(PT:=T#5s),fbTouchGetTap:=(udiMinSingleTapXDiff:=20,udiMinSingleTapYDiff:=20,tMaxDoubleTapTm:=T#900ms,udiMinDoubleTapXDiff:=20,udiMinDoubleTapYDiff:=20),iTablePos:=1,iTablePosTemp:=1); (*Local Variables*)
	END_VAR
END_FUNCTION_BLOCK
```

#### Types.typ - Exported data types
```iecst
TYPE
	tyTouchGetActionInternal : 	STRUCT  (*Local Variables*)
		udiHandle : UDINT; (*Visu Handle*)
		tyTouchAction : TouchAction; (*Output of Touch Action*)
	END_STRUCT;
	tyTouchFilterInternal : 	STRUCT  (*Local Variables*)
		udiXOld : UDINT; (*Old Coordinate X Value*)
		udiYOld : UDINT; (*Old Coordinate Y Value*)
	END_STRUCT;
	tyTouchGetSlideDistInternal : 	STRUCT  (*Local Variables*)
		fbPressedRise : R_TRIG; (*Rising Edge of Press Action*)
		fbInternalPressedRise : R_TRIG; (*Internal Rising Edge of Press Action*)
		bValidStartPress : BOOL; (*Valid of Start Press*)
		bPressed : BOOL; (*Touchscreen Pressed*)
		udiXTemp : UDINT; (*Temporary Coordinate X*)
		udiYTemp : UDINT; (*Temporary Coordinate Y*)
	END_STRUCT;
	tyTouchGetTapInternal : 	STRUCT  (*Local Variables*)
		fbInternalPressedRise : R_TRIG; (*Internal Rising Edge of Press Action*)
		fbInternalPressedFall : F_TRIG; (*Internal Falling Edge of Press Action*)
		bPressed : BOOL; (*Touchscreen Pressed*)
		tTmTemp : TIME; (*Time of Temporary*)
		udiXTemp : UDINT; (*Temporary Coordinate X*)
		udiYTemp : UDINT; (*Temporary Coordinate Y*)
		tTmPrev : TIME; (*Time of Previous*)
		udiXPrev : UDINT; (*Previous Coordinate X*)
		udiYPrev : UDINT; (*Previous Coordinate Y*)
	END_STRUCT;
	tyTableCtrlInternal : 	STRUCT  (*Local Variables*)
		fbSingleTapChkDlyTm : TON; (*Single Tap Check Delay Time*)
		fbSliderOffTm : TON; (*Slider Off Time*)
		fbSelectedRowMnlRise : R_TRIG; (*Rising Edge of Manual Select Row*)
		fbTablePosUpRise : R_TRIG; (*Rising Edge of Up Table Position*)
		fbTablePosDownRise : R_TRIG; (*Rising Edge of Down Table Position*)
		fbSliderRelease : F_TRIG; (*Falling Edge of Slider Active*)
		fbTouchFilter : fbTouchFilter;
		fbTouchGetAction : fbTouchGetAction;
		fbTouchGetSlideDist : fbTouchGetSlideDist;
		fbTouchGetTap : fbTouchGetTap;
		i : INT;
		iTablePos : INT; (*Table Position*)
		iTablePosTemp : INT; (*Temporary Table Position*)
	END_STRUCT;
END_TYPE

(**)
(*Basic Controls*)

TYPE
	tyUILine : 	STRUCT  (*UI Line*)
		uiMaskRtStat : UINT := 1; (*Mask Status Datapoint*)
		uiRtStat : UINT := 0; (*Status Datapoint*)
		usiColor : USINT := 0; (*Color Datapoint*)
	END_STRUCT;
	tyUITxt : 	STRUCT  (*UI Text*)
		bHighlighting : BOOL := FALSE; (*Highlighting Datapoint*)
		sTxt : STRING[30] := ''; (*Text Datapoint*)
		uiMaskRtStat : UINT := 1; (*Mask Status Datapoint*)
		uiRtStat : UINT := 0; (*Status Datapoint*)
		usiColor : USINT := 0; (*Color Datapoint*)
		usiValueIdx : USINT := 0; (*Value Index Datapoint*)
	END_STRUCT;
	tyUIAlmTxt : 	STRUCT  (*UI Text*)
		bHighlighting : BOOL := FALSE; (*Highlighting Datapoint*)
		sTxt : STRING[30] := ''; (*Text Datapoint*)
		uiMaskRtStat : UINT := 1; (*Mask Status Datapoint*)
		uiRtStat : UINT := 0; (*Status Datapoint*)
		usiColor : USINT := 0; (*Color Datapoint*)
		udiValueIdx : UDINT := 0; (*Value Index Datapoint*)
	END_STRUCT;
	tyUIShape : 	STRUCT  (*UI Shape*)
		uiMaskRtStat : UINT := 1; (*Mask Status Datapoint*)
		uiRtStat : UINT := 0; (*Status Datapoint*)
		usiColor : USINT := 0; (*Color Datapoint*)
	END_STRUCT;
	tyUIString : 	STRUCT  (*UI String*)
		bRtCompl : BOOL := FALSE; (*Completion Datapoint*)
		bRtLk : BOOL := FALSE; (*Locking Datapoint*)
		sValue : STRING[30] := ''; (*Value Datapoint*)
		sValueDisplay : STRING[10] := ''; (*Value Datapoint*)
		uiMaskRtStat : UINT := 1; (*Mask Status Datapoint*)
		uiRtStat : UINT := 0; (*Status Datapoint*)
		usiColor : USINT := 0; (*Color Datapoint*)
		sKeypadTitle : STRING[30]; (*Keypad Title*)
	END_STRUCT;
	tyUILString : 	STRUCT  (*UI String*)
		bRtCompl : BOOL := FALSE; (*Completion Datapoint*)
		bRtLk : BOOL := FALSE; (*Locking Datapoint*)
		sValue : STRING[254] := ''; (*Value Datapoint*)
		uiMaskRtStat : UINT := 1; (*Mask Status Datapoint*)
		uiRtStat : UINT := 0; (*Status Datapoint*)
		usiColor : USINT := 0; (*Color Datapoint*)
		sKeypadTitle : STRING[30]; (*Keypad Title*)
	END_STRUCT;
	tyUINum : 	STRUCT  (*UI Numeric*)
		bRtCompl : BOOL := FALSE; (*Completion Datapoint*)
		bRtLk : BOOL := FALSE; (*Locking Datapoint*)
		diValue : DINT := 0; (*Value Datapoint*)
		diValueMax : DINT := 0; (*Max Value Datapoint*)
		diValueMin : DINT := 0; (*Min Value Datapoint*)
		diValueTeach : DINT := 0; (*Teach Value Datapoint*)
		uiMaskRtStat : UINT := 1; (*Mask Status Datapoint*)
		uiRtStat : UINT := 0; (*Status Datapoint*)
		usiAddDigits : USINT := 0; (*Add Fraction Digits Datapoint*)
		usiColor : USINT := 0; (*Color Datapoint*)
		sKeypadTitle : STRING[30]; (*Keypad Title*)
	END_STRUCT;
	tyUIBtn : 	STRUCT  (*UI Button*)
		bRtCompl : BOOL := FALSE; (*Completion Datapoint*)
		bRtLk : BOOL := FALSE; (*Locking Datapoint*)
		bValue : BOOL := FALSE; (*Boolean Value Datapoint*)
		uiMaskRtStat : UINT := 1; (*Mask Status Datapoint*)
		uiRtStat : UINT := 0; (*Status Datapoint*)
		usiBitmapIdx : USINT := 0; (*Bitmap Index Datapoint*)
		usiColor : USINT := 0; (*Color Datapoint*)
		usiPressedColor : USINT := 0; (*Button Pressed Color Datapoint*)
		usiTxtIdx : USINT := 0; (*Text Index Datapoint*)
		uiBitmapIdx : UINT := 0; (*Bitmap Index Datapoint*)
	END_STRUCT;
	tyUIHotspot : 	STRUCT  (*UI Hotspot*)
		bRtCompl : BOOL := FALSE; (*Completion Datapoint*)
		bRtLk : BOOL := FALSE; (*Locking Datapoint*)
		bValue : BOOL := FALSE; (*Boolean Value Datapoint*)
		uiMaskRtStat : UINT := 1; (*Mask Status Datapoint*)
		uiRtStat : UINT := 0; (*Status Datapoint*)
	END_STRUCT;
	tyUIBitmap : 	STRUCT  (*UI Bitmap*)
		uiMaskRtStat : UINT := 1; (*Mask Status Datapoint*)
		uiRtStat : UINT := 0; (*Status Datapoint*)
		usiColor : USINT := 0; (*Color Datapoint*)
		usiValueIdx : USINT := 0; (*Value Index Datapoint*)
		uiValueIdx : UINT := 0; (*Value Index Datapoint*)
	END_STRUCT;
	tyUIBarGraph : 	STRUCT  (*UI Bar Graph*)
		iValue : INT := 0; (*Value Datapoint*)
		uiMaskRtStat : UINT := 1; (*Mask Status Datapoint*)
		uiRtStat : UINT := 0; (*Status Datapoint*)
		usiColor : USINT := 0; (*Color Datapoint*)
	END_STRUCT;
	tyUIDT : 	STRUCT  (*UI DateTime*)
		diValue : DINT := 0; (*Value Datapoint*)
		uiMaskRtStat : UINT := 1; (*Mask Status Datapoint*)
		uiRtStat : UINT := 0; (*Status Datapoint*)
		usiColor : USINT := 0; (*Color Datapoint*)
	END_STRUCT;
	tyUIPw : 	STRUCT  (*UI Password*)
		a_sTxt : ARRAY[0..9]OF STRING[30] := [10('')]; (*Text Datapoint*)
		bRtCompl : BOOL := FALSE; (*Completion Datapoint*)
		bRtLk : BOOL := FALSE; (*Locking Datapoint*)
		uiMaskRtStat : UINT := 1; (*Mask Status Datapoint*)
		uiRtStat : UINT := 0; (*Status Datapoint*)
		usiColor : USINT := 0; (*Color Datapoint*)
		usiLevel : USINT := 0; (*Level Datapoint*)
	END_STRUCT;
	tyUIListBox : 	STRUCT  (*UI List Box*)
		a_sTxt : ARRAY[0..9]OF STRING[30] := [10('')]; (*Text Datapoint*)
		a_usiValueOptionIdx : ARRAY[0..9]OF USINT := [10(0)]; (*Option Value Index Datapoint*)
		bRtCompl : BOOL := FALSE; (*Completion Datapoint*)
		bRtLk : BOOL := FALSE; (*Locking Datapoint*)
		uiMaskRtStat : UINT := 1; (*Mask Status Datapoint*)
		uiRtStat : UINT := 0; (*Status Datapoint*)
		usiColor : USINT := 0; (*Color Datapoint*)
		usiDisabledColor : USINT := 0; (*Disabled Color Datapoint*)
		usiSelectedColor : USINT := 0; (*Selected Color Datapoint*)
		usiSliderColor : USINT := 0; (*Slider Color Datapoint*)
		usiValueIdx : USINT := 0; (*Value Index Datapoint*)
		usiValueMaxIdx : USINT := 0; (*Max Value Index Datapoint*)
		usiValueMinIdx : USINT := 0; (*Min Value Index Datapoint*)
	END_STRUCT;
	tyUIAlm : 	STRUCT  (*UI Alarm*)
		a_usiFltrTm : ARRAY[0..5]OF USINT := [6(0)]; (*Filter Time Datapoint*)
		bRtLk : BOOL := FALSE; (*Locking Datapoint*)
		uiMaskRtStat : UINT := 1; (*Mask Status Datapoint*)
		uiRtStat : UINT := 0; (*Status Datapoint*)
		usiColor : USINT := 0; (*Color Datapoint*)
		uiFltrAlm : UINT := 0; (*Filter Alarm Datapoint*)
		uiFltrCtrl : UINT := 0; (*Filter Control Datapoint*)
		uiFltrGrp : UINT := 0; (*Filter Group Datapoint*)
		uiFltrPriority : UINT := 0; (*Filter Priority Datapoint*)
	END_STRUCT;
	tyUIDrawBox : 	STRUCT  (*UI Draw Box*)
		uiMaskRtStat : UINT := 1; (*Mask Status Datapoint*)
		uiRtStat : UINT := 0; (*Status Datapoint*)
	END_STRUCT;
	tyUITrend : 	STRUCT  (*UI Trend*)
		bRtCompl : BOOL := FALSE; (*Completion Datapoint*)
		bRtLk : BOOL := FALSE; (*Locking Datapoint*)
		iSelectItem : INT := 0; (*Select Item Datapoint*)
		uiMaskRtStat : UINT := 1; (*Mask Status Datapoint*)
		uiRtStat : UINT := 0; (*Status Datapoint*)
		usiColor : USINT := 0; (*Color Datapoint*)
	END_STRUCT;
	tyUIScale : 	STRUCT  (*UI Scale*)
		iMaxValue : INT := 0; (*Max Value Datapoint*)
		iMinValue : INT := 0; (*Min Value Datapoint*)
		iRangeEnd : INT := 0; (*Range End Datapoint*)
		iRangeSt : INT := 0; (*Range Start Datapoint*)
		iValue : INT := 0; (*Value Datapoint*)
		uiMaskRtStat : UINT := 1; (*Mask Status Datapoint*)
		uiRtStat : UINT := 0; (*Status Datapoint*)
		usiColor : USINT := 0; (*Color Datapoint*)
		usiRangeColor : USINT := 0; (*Range Color Datapoint*)
	END_STRUCT;
	tyUIEdit : 	STRUCT  (*UI Edit*)
		bLineEndings : BOOL := FALSE; (*Line Endings Datapoint*)
		bRtCompl : BOOL := FALSE; (*Completion Datapoint*)
		bRtEditInsertMode : BOOL := FALSE; (*Edit Insert Mode Datapoint*)
		bRtEditModified : BOOL := FALSE; (*Edit Modified Datapoint*)
		bRtEditSelectionMode : BOOL := FALSE; (*Edit Selection Mode Datapoint*)
		bRtLk : BOOL := FALSE; (*Locking Datapoint*)
		iRtEditCursorColumn : INT := 0; (*Edit Cursor Column Datapoint*)
		iRtEditCursorLine : INT := 0; (*Edit Cursor Line Datapoint*)
		sRtCmdRequest : STRING[30] := ''; (*Command Request Datapoint*)
		sRtCmdResponse : STRING[30] := ''; (*Command Response Datapoint*)
		sURL : STRING[30] := ''; (*URL Datapoint*)
		sValue : STRING[30] := ''; (*Value Datapoint*)
		uiMaskRtStat : UINT := 1; (*Mask Status Datapoint*)
		uiRtBusy : UINT := 0; (*Busy Datapoint*)
		uiRtCmdStat : UINT := 0; (*Command Status Datapoint*)
		uiRtStat : UINT := 0; (*Status Datapoint*)
		usiColor : USINT := 0; (*Color Datapoint*)
		usiCursorColor : USINT := 0; (*Cursor Color Datapoint*)
		usiSelectedColor : USINT := 0; (*Selected Color Datapoint*)
	END_STRUCT;
	tyUIHTMLView : 	STRUCT  (*UI HTML View*)
		bRtLk : BOOL := FALSE; (*Locking Datapoint*)
		sChgURL : STRING[30] := ''; (*Change URL Datapoint*)
		sCurrTitle : STRING[30] := ''; (*Current Title Datapoint*)
		sCurrURL : STRING[30] := ''; (*Current URL Datapoint*)
		sHTMLStream : STRING[30] := ''; (*HTML Stream*)
		uiMaskRtStat : UINT := 1; (*Mask Status Datapoint*)
		uiRtBusy : UINT := 0; (*Busy Datapoint*)
		uiRtHTTPErrCode : UINT := 0; (*HTTP Error Code*)
		uiRtStat : UINT := 0; (*Status Datapoint*)
		usiColor : USINT := 0; (*Color Datapoint*)
		usiErrCnt : USINT := 0; (*Error Count Datapoint*)
	END_STRUCT;
	tyUIDrpDn : 	STRUCT  (*UI Dropdown*)
		a_usiValueOptionIdx : ARRAY[0..9]OF USINT := [10(0)]; (*Option Value Index Datapoint*)
		bRtCompl : BOOL := FALSE; (*Completion Datapoint*)
		bRtLk : BOOL := FALSE; (*Locking Datapoint*)
		sTxt : STRING[30] := ''; (*Text Datapoint*)
		uiMaskRtStat : UINT := 1; (*Mask Status Datapoint*)
		uiRtStat : UINT := 0; (*Status Datapoint*)
		usiColor : USINT := 0; (*Color Datapoint*)
		usiDisabledColor : USINT := 0; (*Disabled Color Datapoint*)
		usiDropdownColor : USINT := 0; (*Dropdown Color Datapoint*)
		usiSelectedColor : USINT := 0; (*Selected Color Datapoint*)
		usiValueIdx : USINT := 0; (*Value Index Datapoint*)
		usiValueMaxIdx : USINT := 0; (*Max Value Index Datapoint*)
		usiValueMinIdx : USINT := 0; (*Min Value Index Datapoint*)
	END_STRUCT;
	tyUIPieChart : 	STRUCT  (*UI Pie Chart*)
		a_uiValue : ARRAY[0..9]OF UINT := [10(0)]; (*Value Datapoint*)
		uiMaskRtStat : UINT := 1; (*Mask Status Datapoint*)
		uiRtStat : UINT := 0; (*Status Datapoint*)
		usiColor : USINT := 0; (*Color Datapoint*)
	END_STRUCT;
	tyUISlider : 	STRUCT  (*UI Slider*)
		bRtCompl : BOOL := FALSE; (*Completion Datapoint*)
		bRtLk : BOOL := FALSE; (*Locking Datapoint*)
		iCurrValue : INT := 0; (*Current Value Datapoint*)
		iMaxValue : INT := 0; (*Max Value Datapoint*)
		iMinValue : INT := 0; (*Min Value Datapoint*)
		iValue : INT := 0; (*Value Datapoint*)
		uiMaskRtStat : UINT := 1; (*Mask Status Datapoint*)
		uiRtStat : UINT := 0; (*Status Datapoint*)
		usiColor : USINT := 0; (*Color Datapoint*)
	END_STRUCT;
	tyUIGauge : 	STRUCT  (*UI Gauge*)
		iMaxValue : INT := 0; (*Max Value Datapoint*)
		iMinValue : INT := 0; (*Min Value Datapoint*)
		iValue : INT := 0; (*Value Datapoint*)
		uiMaskRtStat : UINT := 1; (*Mask Status Datapoint*)
		uiRtStat : UINT := 0; (*Status Datapoint*)
		usiColor : USINT := 0; (*Color Datapoint*)
	END_STRUCT;
	tyUITable : 	STRUCT  (*UI Table*)
		a_tyHotspot : ARRAY[1..15]OF tyUIHotspot; (*Array Of Hotspot*)
		a_tyStringDataCol0 : ARRAY[1..15]OF tyUILString; (*Array Of Number Listing (column: 0 / x = 0)*)
		a_tyStringDataCol1 : ARRAY[1..15]OF tyUILString; (*Array Of Data (column: 1 / x = 1)*)
		a_tyStringDataCol2 : ARRAY[1..15]OF tyUILString; (*Array Of Data (column: 2 / x = 2)*)
		a_tyStringDataCol3 : ARRAY[1..15]OF tyUILString; (*Array Of Data (column: 3 / x = 3)*)
		a_tyStringDataCol4 : ARRAY[1..15]OF tyUILString; (*Array Of Data (column: 4 / x = 4)*)
		tyUISlider : tyUISlider := (uiRtStat:=1); (*Scroll Bar Scale*)
		tyStringTitle0Col0Row0 : tyUIString; (*Number Listing Title (row: 0, column: 0 / x = 0, y = 0)*)
		tyStringTitle1Col1Row0 : tyUIString; (*Title (row: 0, column: 1 / x = 1, y = 0)*)
		tyStringTitle2Col2Row0 : tyUIString; (*Title (row: 0, column: 2 / x = 2, y = 0)*)
		tyStringTitle3Col3Row0 : tyUIString; (*Title (row: 0, column: 3 / x = 3, y = 0)*)
		tyStringTitle4Col4Row0 : tyUIString; (*Title (row: 0, column: 4 / x = 4, y = 0)*)
		uiMaskRtStat : UINT := 1; (*Mask Status Datapoint*)
	END_STRUCT;
	tyUITable1 : 	STRUCT  (*UI Table*)
		a_tyHotspot : ARRAY[1..15]OF tyUIHotspot; (*Array Of Hotspot*)
		a_tyStringDataCol0 : ARRAY[1..15]OF tyUILString; (*Array Of Number Listing (column: 0 / x = 0)*)
		a_tyStringDataCol1 : ARRAY[1..15]OF tyUILString; (*Array Of Data (column: 1 / x = 1)*)
		a_tyStringDataCol2 : ARRAY[1..15]OF tyUILString; (*Array Of Data (column: 2 / x = 2)*)
		a_tyStringDataCol4 : ARRAY[1..15]OF tyUILString; (*Array Of Data (column: 4 / x = 4)*)
		a_tyTxtDataCol3 : ARRAY[1..15]OF tyUITxt; (*Array Of Data (column: 3 / x = 3)*)
		tyStringTitle0Col0Row0 : tyUIString; (*Number Listing Title (row: 0, column: 0 / x = 0, y = 0)*)
		tyStringTitle1Col1Row0 : tyUIString; (*Title (row: 0, column: 1 / x = 1, y = 0)*)
		tyStringTitle2Col2Row0 : tyUIString; (*Title (row: 0, column: 2 / x = 2, y = 0)*)
		tyStringTitle3Col3Row0 : tyUIString; (*Title (row: 0, column: 3 / x = 3, y = 0)*)
		tyStringTitle4Col4Row0 : tyUIString; (*Title (row: 0, column: 4 / x = 4, y = 0)*)
		tyUISlider : tyUISlider := (uiRtStat:=1); (*Scroll Bar Scale*)
		uiMaskRtStat : UINT := 1; (*Mask Status Datapoint*)
	END_STRUCT;
	tyUILyr : 	STRUCT  (*UI Layer*)
		uiRtStat : UINT := 0; (*Status Datapoint*)
	END_STRUCT;
	tyUIAlarm : 	STRUCT
		tyUIAlmCur : tyAlm;
		tyUIAlmHis : tyAlm;
	END_STRUCT;
	tyAlm : 	STRUCT
		usiColor : USINT;
		udiCntrllDp : INT;
		udiGrpDp : UDINT;
		udiAlrmDp : UDINT;
		udiPrioDp : UDINT;
		udiTimeDp : DATE_AND_TIME;
		uiRtStat : UINT;
	END_STRUCT;
	tyUIAlarmInfoGrp : 	STRUCT
		udiOffsetInfo1 : UDINT;
		udiOffsetInfo2 : UDINT;
		tyUptTxtSnipp : tyUIAlmTextSnip;
		udiToggleAlarmInfo : UDINT;
	END_STRUCT;
	tyUIAlmTextSnip : 	STRUCT
		CurrentRecipeName : STRING[80];
		CurrentRecipeWidth : STRING[80];
		SameRcpDiffWidName : STRING[80];
		MachineOutGoingWidth : STRING[80];
		LFNewRecipeName : STRING[80];
		LFNewRecipeWidth : STRING[80];
		LFOldRecipeName : STRING[80];
		LFOldRecipeWidth : STRING[80];
		HANewRecipeName : STRING[80];
		HANewRecipeWidth : STRING[80];
		HAOldRecipeName : STRING[80];
		HAOldRecipeWidth : STRING[80];
		HBNewRecipeName : STRING[80];
		HBNewRecipeWidth : STRING[80];
		HBOldRecipeName : STRING[80];
		HBOldRecipeWidth : STRING[80];
	END_STRUCT;
END_TYPE
```

#### fUIInRtStatLock.st
```iecst
(* Runtime Status Datapoint Lock *)
FUNCTION fUIInRtStatLock

	uiRtStat.0		:= FALSE;
	uiRtStat.1		:= TRUE;
	uiRtStat.2		:= FALSE;
	uiRtStat.3		:= FALSE;

	fUIInRtStatLock	:= uiRtStat;

END_FUNCTION
```

#### fUIInRtStatHide.st
```iecst
(* Runtime Status Datapoint Lock *)
FUNCTION fUIInRtStatHide

	uiRtStat.0		:= TRUE;
	uiRtStat.1		:= FALSE;
	uiRtStat.2		:= FALSE;
	uiRtStat.3		:= FALSE;

	fUIInRtStatHide	:= uiRtStat;

END_FUNCTION
```

#### fUIInRtStatFocus.st
```iecst
(* Runtime Status Datapoint Lock *)
FUNCTION fUIInRtStatFocus

	uiRtStat.0			:= FALSE;
	uiRtStat.1			:= FALSE;
	uiRtStat.2			:= TRUE;
	uiRtStat.3			:= FALSE;

	fUIInRtStatFocus	:= uiRtStat;

END_FUNCTION
```

#### fUIOutRtStatCursor1Valid.st
```iecst
(* Runtime Status Datapoint Lock *)
FUNCTION fUIOutRtStatCursor1Valid

	fUIOutRtStatCursor1Valid	:= uiRtStat.10;

END_FUNCTION
```

#### fUIInRtStatOpenTP.st
```iecst
(* Runtime Status Datapoint Lock *)
FUNCTION fUIInRtStatOpenTP

	uiRtStat.0			:= FALSE;
	uiRtStat.1			:= FALSE;
	uiRtStat.2			:= FALSE;
	uiRtStat.3			:= TRUE;

	fUIInRtStatOpenTP	:= uiRtStat;

END_FUNCTION
```

#### fUIOutRtStatCursor2Valid.st
```iecst
(* Runtime Status Datapoint Lock *)
FUNCTION fUIOutRtStatCursor2Valid

	fUIOutRtStatCursor2Valid	:= uiRtStat.11;

END_FUNCTION
```

#### fUIOutRtStatHasFocus.st
```iecst
(* Runtime Status Datapoint Lock *)
FUNCTION fUIOutRtStatHasFocus

	fUIOutRtStatHasFocus	:= uiRtStat.14;

END_FUNCTION
```

#### fUIInRtStatOff.st
```iecst
(* Runtime Status Datapoint Lock *)
FUNCTION fUIInRtStatOff

	uiRtStat.0		:= FALSE;
	uiRtStat.1		:= FALSE;
	uiRtStat.2		:= FALSE;
	uiRtStat.3		:= FALSE;

	fUIInRtStatOff	:= uiRtStat;

END_FUNCTION
```

#### fUIOutRtStatInEdit.st
```iecst
(* Runtime Status Datapoint Lock *)
FUNCTION fUIOutRtStatInEdit

	fUIOutRtStatInEdit	:= uiRtStat.15;

END_FUNCTION
```

#### fUIOutRtStatOnLock.st
```iecst
(* Runtime Status Datapoint Lock *)
FUNCTION fUIOutRtStatOnLock

	fUIOutRtStatOnLock	:= uiRtStat.13;

END_FUNCTION
```

#### fUIOutRtStatTPIsOpen.st
```iecst
(* Runtime Status Datapoint Lock *)
FUNCTION fUIOutRtStatTPIsOpen

	fUIOutRtStatTPIsOpen	:= uiRtStat.12;

END_FUNCTION
```

#### fbTouchGetAction.st
```iecst
(* Get Touch Action Coordinate *)
FUNCTION_BLOCK fbTouchGetAction

	IF tyInternal.udiHandle = 0 THEN
		tyInternal.udiHandle	:= VA_Setup(TRUE , sVisuNm);

	ELSE
		IF VA_Saccess(TRUE , tyInternal.udiHandle) = 0 THEN
			VA_GetTouchAction(TRUE , tyInternal.udiHandle , 0 , ADR(tyInternal.tyTouchAction));

			bPressed	:= tyInternal.tyTouchAction.status = 1;
			udiX		:= tyInternal.tyTouchAction.x;
			udiY		:= tyInternal.tyTouchAction.y;

			VA_Srelease(TRUE ,tyInternal.udiHandle);

		END_IF

	END_IF

END_FUNCTION_BLOCK
```

#### fbTouchGetSlideDist.st
```iecst
(* Get Slide Distance *)
FUNCTION_BLOCK fbTouchGetSlideDist

	//Get Valid Press
	tyInternal.fbPressedRise(CLK := bPressed);

	IF tyInternal.fbPressedRise.Q THEN
		IF udiX > udiWorkAreaStartX AND udiX < udiWorkAreaEndX AND udiY > udiWorkAreaStartY AND udiY < udiWorkAreaEndY THEN
			tyInternal.bValidStartPress	:= TRUE;
		ELSE
			tyInternal.bValidStartPress	:= FALSE;
		END_IF
	END_IF

	IF bPressed AND tyInternal.bValidStartPress THEN
		tyInternal.bPressed	:= TRUE;
	ELSE
		tyInternal.bPressed	:= FALSE;
	END_IF

	//Update Press Record
	tyInternal.fbInternalPressedRise(CLK := tyInternal.bPressed);

	IF tyInternal.fbInternalPressedRise.Q THEN
		tyInternal.udiXTemp	:= udiX;
		tyInternal.udiYTemp	:= udiY;

	END_IF

	//Get Valid Press Coordinate
	IF tyInternal.bPressed = TRUE THEN
		diXDist	:= UDINT_TO_DINT(udiX) - UDINT_TO_DINT(tyInternal.udiXTemp);
		diYDist	:= UDINT_TO_DINT(udiY) - UDINT_TO_DINT(tyInternal.udiYTemp);

		IF DINT_TO_UDINT(ABS(diXDist)) < udiMinXDist THEN
			diXDist	:= 0;
		END_IF

		IF DINT_TO_UDINT(ABS(diYDist)) < udiMinYDist THEN
			diYDist	:= 0;
		END_IF

	ELSE
		diXDist	:= 0;
		diYDist	:= 0;

	END_IF

END_FUNCTION_BLOCK
```

#### fbTouchGetTap.st
```iecst
(* Get Double Tap *)
FUNCTION_BLOCK fbTouchGetTap

	IF bPressed AND udiX > udiWorkAreaStartX AND udiX < udiWorkAreaEndX AND udiY > udiWorkAreaStartY AND udiY < udiWorkAreaEndY THEN
		tyInternal.bPressed	:= TRUE;
	ELSE
		tyInternal.bPressed	:= FALSE;
	END_IF

	tyInternal.fbInternalPressedRise(CLK := tyInternal.bPressed);
	tyInternal.fbInternalPressedFall(CLK := tyInternal.bPressed);

	IF tyInternal.fbInternalPressedRise.Q THEN
		tyInternal.tTmTemp	:= clock_ms();
		tyInternal.udiXTemp	:= udiX;
		tyInternal.udiYTemp	:= udiY;

		bSingleTap		:= FALSE;
		udiSingleTapX	:= 0;
		udiSingleTapY	:= 0;

		bDoubleTap		:= FALSE;
		udiDoubleTapX	:= 0;
		udiDoubleTapY	:= 0;

	ELSIF tyInternal.fbInternalPressedFall.Q THEN
		IF ((clock_ms() - tyInternal.tTmPrev) < tMaxDoubleTapTm) AND (ABS(UDINT_TO_DINT(udiX) - UDINT_TO_DINT(tyInternal.udiXPrev)) < UDINT_TO_DINT(udiMinDoubleTapXDiff)) AND (ABS(UDINT_TO_DINT(udiY) - UDINT_TO_DINT(tyInternal.udiYPrev)) < UDINT_TO_DINT(udiMinDoubleTapYDiff)) THEN
			bDoubleTap		:= TRUE;
			udiDoubleTapX	:= (udiX + tyInternal.udiXPrev) / 2;
			udiDoubleTapY	:= (udiY + tyInternal.udiYPrev) / 2;

		END_IF

		IF (ABS(UDINT_TO_DINT(udiX) - UDINT_TO_DINT(tyInternal.udiXTemp)) < UDINT_TO_DINT(udiMinSingleTapXDiff)) AND (ABS(UDINT_TO_DINT(udiY) - UDINT_TO_DINT(tyInternal.udiYTemp)) < UDINT_TO_DINT(udiMinSingleTapYDiff)) THEN
			bSingleTap		:= TRUE;
			udiSingleTapX	:= tyInternal.udiXTemp;
			udiSingleTapY	:= tyInternal.udiYTemp;

		END_IF

		tyInternal.tTmPrev	:= tyInternal.tTmTemp;
		tyInternal.udiXPrev	:= tyInternal.udiXTemp;
		tyInternal.udiYPrev	:= tyInternal.udiYTemp;

	END_IF

END_FUNCTION_BLOCK
```

#### fbTableCtrl.st
```iecst
(* Table Control *)
FUNCTION_BLOCK fbTableCtrl

	bSliderActive	:= FALSE;

	FOR tyInternal.i := 1 TO 15 DO
		IF a_tyUIHotspot[tyInternal.i].bRtCompl THEN
			bTableActive	:= TRUE;
		END_IF

	END_FOR

	tyInternal.fbSliderRelease(CLK := uiSliderStatus.15);

	IF uiSliderStatus.15 THEN
		tyInternal.fbSliderOffTm(IN := FALSE);

		tyInternal.iTablePos	:= iSliderPos;

		IF tyInternal.iTablePos > (iTotalData - iTotalRow + 1) THEN
			IF (iTotalData - iTotalRow + 1) < 1 THEN
				tyInternal.iTablePos	:= 1;
			ELSE
				tyInternal.iTablePos	:= iTotalData - iTotalRow + 1;
			END_IF

		ELSIF tyInternal.iTablePos < 1 THEN
			tyInternal.iTablePos	:= 1;

		END_IF

		uiTablePos	:= INT_TO_UINT(tyInternal.iTablePos);
		iSliderPos	:= UINT_TO_INT(uiTablePos);

		tyInternal.iTablePosTemp	:= UINT_TO_INT(uiTablePos);

		bSliderActive	:= TRUE;

	ELSIF tyInternal.fbSliderRelease.Q = TRUE THEN
		bSliderActive	:= TRUE;
		iSliderPos		:= UINT_TO_INT(uiTablePos);

	ELSIF bTableActive THEN
		//Get Touch Coordinate
		tyInternal.fbTouchGetAction.sVisuNm	:= sVisuNm;
		tyInternal.fbTouchGetAction;

		//Touch Filter
		tyInternal.fbTouchFilter.bPressedIn	:= tyInternal.fbTouchGetAction.bPressed;
		tyInternal.fbTouchFilter.udiXIn		:= tyInternal.fbTouchGetAction.udiX;
		tyInternal.fbTouchFilter.udiYIn		:= tyInternal.fbTouchGetAction.udiY;
		tyInternal.fbTouchFilter;

		//Get Slide Function Block
		tyInternal.fbTouchGetSlideDist.udiWorkAreaStartX	:= udiWorkAreaStartX;
		tyInternal.fbTouchGetSlideDist.udiWorkAreaStartY	:= udiWorkAreaStartY;
		tyInternal.fbTouchGetSlideDist.udiWorkAreaEndX		:= udiWorkAreaEndX;
		tyInternal.fbTouchGetSlideDist.udiWorkAreaEndY		:= udiWorkAreaEndY;
		tyInternal.fbTouchGetSlideDist.udiMinXDist			:= udiMinXDist;
		tyInternal.fbTouchGetSlideDist.udiMinYDist			:= udiMinYDist;
		tyInternal.fbTouchGetSlideDist.bPressed				:= tyInternal.fbTouchFilter.bPressedOut;
		tyInternal.fbTouchGetSlideDist.udiX					:= tyInternal.fbTouchFilter.udiXOut;
		tyInternal.fbTouchGetSlideDist.udiY					:= tyInternal.fbTouchFilter.udiYOut;
		tyInternal.fbTouchGetSlideDist;

		//Get Tap Function Block
		tyInternal.fbTouchGetTap.udiWorkAreaStartX		:= udiWorkAreaStartX;
		tyInternal.fbTouchGetTap.udiWorkAreaStartY		:= udiWorkAreaStartY;
		tyInternal.fbTouchGetTap.udiWorkAreaEndX		:= udiWorkAreaEndX;
		tyInternal.fbTouchGetTap.udiWorkAreaEndY		:= udiWorkAreaEndY;
		tyInternal.fbTouchGetTap.udiMinSingleTapXDiff	:= udiMinXDist;
		tyInternal.fbTouchGetTap.udiMinSingleTapYDiff	:= udiMinYDist;
		tyInternal.fbTouchGetTap.bPressed				:= tyInternal.fbTouchFilter.bPressedOut;
		tyInternal.fbTouchGetTap.udiX					:= tyInternal.fbTouchFilter.udiXOut;
		tyInternal.fbTouchGetTap.udiY					:= tyInternal.fbTouchFilter.udiYOut;
		tyInternal.fbTouchGetTap;

		fUIInRtStatOff(ADR(uiSliderStatus));

		IF tyInternal.fbTouchFilter.bPressedOut = TRUE THEN
			tyInternal.fbSliderOffTm(IN := FALSE);
			tyInternal.fbSingleTapChkDlyTm(IN := FALSE);

			IF uiSlideScale < 1 THEN
				uiSlideScale	:= 1;
			END_IF

			tyInternal.iTablePos	:= tyInternal.iTablePosTemp - DINT_TO_INT(tyInternal.fbTouchGetSlideDist.diYDist) / UINT_TO_INT(uiSlideScale);

			IF tyInternal.iTablePos > (iTotalData - iTotalRow + 1) THEN
				IF (iTotalData - iTotalRow + 1) < 1 THEN
					tyInternal.iTablePos	:= 1;
				ELSE
					tyInternal.iTablePos	:= iTotalData - iTotalRow + 1;
				END_IF

			ELSIF tyInternal.iTablePos < 1 THEN
				tyInternal.iTablePos	:= 1;

			END_IF

			uiTablePos	:= INT_TO_UINT(tyInternal.iTablePos);
			iSliderPos	:= UINT_TO_INT(uiTablePos);

		ELSE
			tyInternal.iTablePosTemp	:= tyInternal.iTablePos;

			tyInternal.fbSingleTapChkDlyTm(IN := TRUE);

			IF tyInternal.fbSingleTapChkDlyTm.Q = TRUE THEN
				FOR tyInternal.i := 1 TO 15 DO
					a_tyUIHotspot[tyInternal.i].bRtCompl	:= FALSE;
				END_FOR

				bTableActive	:= FALSE;

			ELSE
				FOR tyInternal.i := 1 TO 15 DO
					IF a_tyUIHotspot[tyInternal.i].bValue = TRUE THEN
						IF tyInternal.fbTouchGetTap.bSingleTap = TRUE THEN
							uiSelectedRow	:= tyInternal.i;
						END_IF

						a_tyUIHotspot[tyInternal.i].bValue	:= FALSE;

					END_IF

				END_FOR

			END_IF

		END_IF

	ELSIF uiSliderStatus.0 = FALSE THEN
		tyInternal.fbSliderOffTm(IN := TRUE);

		IF tyInternal.fbSliderOffTm.Q = TRUE THEN
			fUIInRtStatHide(ADR(uiSliderStatus));
			tyInternal.fbSliderOffTm(IN := FALSE);

		END_IF

	END_IF

	tyInternal.fbSelectedRowMnlRise(CLK := bSelectedRowMnl);
	IF tyInternal.fbSelectedRowMnlRise.Q THEN
		uiSelectedRow	:= uiSelectedRowMnl;
	END_IF

	tyInternal.fbTablePosUpRise(CLK := bTablePosPlus);
	IF tyInternal.fbTablePosUpRise.Q THEN
		uiTablePos					:= uiTablePos + 1;
		iSliderPos					:= iSliderPos + 1;
		tyInternal.iTablePos		:= tyInternal.iTablePos + 1;
		tyInternal.iTablePosTemp	:= tyInternal.iTablePosTemp + 1;

	END_IF

	tyInternal.fbTablePosDownRise(CLK := bTablePosMinus);
	IF tyInternal.fbTablePosDownRise.Q THEN
		uiTablePos					:= uiTablePos - 1;
		iSliderPos					:= iSliderPos - 1;
		tyInternal.iTablePos		:= tyInternal.iTablePos - 1;
		tyInternal.iTablePosTemp	:= tyInternal.iTablePosTemp - 1;

	END_IF

END_FUNCTION_BLOCK
```

#### fbTableCtrl_v2.st
```iecst
(* Table Control Version 2 *)
FUNCTION_BLOCK fbTableCtrl_v2

	p_bSliderActive	:= FALSE;

	FOR tyInternal.i := 1 TO 15 DO
		IF pa_tyUIHotspot[tyInternal.i].bRtCompl THEN
			p_bTableActive	:= TRUE;
		END_IF

	END_FOR

	tyInternal.fbSliderRelease(CLK := p_uiSliderStatus.15);

	IF p_uiSliderStatus.15 THEN
		tyInternal.fbSliderOffTm(IN := FALSE);

		tyInternal.iTablePos	:= p_iSliderPos;

		IF tyInternal.iTablePos > (iTotalData - iTotalRow + 1) THEN
			IF (iTotalData - iTotalRow + 1) < 1 THEN
				tyInternal.iTablePos	:= 1;
			ELSE
				tyInternal.iTablePos	:= iTotalData - iTotalRow + 1;
			END_IF

		ELSIF tyInternal.iTablePos < 1 THEN
			tyInternal.iTablePos	:= 1;

		END_IF

		p_uiTablePos	:= INT_TO_UINT(tyInternal.iTablePos);
		p_iSliderPos	:= UINT_TO_INT(p_uiTablePos);

		tyInternal.iTablePosTemp	:= UINT_TO_INT(p_uiTablePos);

		p_bSliderActive	:= TRUE;

	ELSIF tyInternal.fbSliderRelease.Q = TRUE THEN
		p_bSliderActive	:= TRUE;
		p_iSliderPos	:= UINT_TO_INT(p_uiTablePos);

	ELSIF p_bTableActive THEN
		//Get Touch Coordinate
		tyInternal.fbTouchGetAction.sVisuNm	:= sVisuNm;
		tyInternal.fbTouchGetAction;

		//Touch Filter
		tyInternal.fbTouchFilter.bPressedIn	:= tyInternal.fbTouchGetAction.bPressed;
		tyInternal.fbTouchFilter.udiXIn		:= tyInternal.fbTouchGetAction.udiX;
		tyInternal.fbTouchFilter.udiYIn		:= tyInternal.fbTouchGetAction.udiY;
		tyInternal.fbTouchFilter;

		//Get Slide Function Block
		tyInternal.fbTouchGetSlideDist.udiWorkAreaStartX	:= udiWorkAreaStartX;
		tyInternal.fbTouchGetSlideDist.udiWorkAreaStartY	:= udiWorkAreaStartY;
		tyInternal.fbTouchGetSlideDist.udiWorkAreaEndX		:= udiWorkAreaEndX;
		tyInternal.fbTouchGetSlideDist.udiWorkAreaEndY		:= udiWorkAreaEndY;
		tyInternal.fbTouchGetSlideDist.udiMinXDist			:= udiMinXDist;
		tyInternal.fbTouchGetSlideDist.udiMinYDist			:= udiMinYDist;
		tyInternal.fbTouchGetSlideDist.bPressed				:= tyInternal.fbTouchFilter.bPressedOut;
		tyInternal.fbTouchGetSlideDist.udiX					:= tyInternal.fbTouchFilter.udiXOut;
		tyInternal.fbTouchGetSlideDist.udiY					:= tyInternal.fbTouchFilter.udiYOut;
		tyInternal.fbTouchGetSlideDist;

		//Get Tap Function Block
		tyInternal.fbTouchGetTap.udiWorkAreaStartX		:= udiWorkAreaStartX;
		tyInternal.fbTouchGetTap.udiWorkAreaStartY		:= udiWorkAreaStartY;
		tyInternal.fbTouchGetTap.udiWorkAreaEndX		:= udiWorkAreaEndX;
		tyInternal.fbTouchGetTap.udiWorkAreaEndY		:= udiWorkAreaEndY;
		tyInternal.fbTouchGetTap.udiMinSingleTapXDiff	:= udiMinXDist;
		tyInternal.fbTouchGetTap.udiMinSingleTapYDiff	:= udiMinYDist;
		tyInternal.fbTouchGetTap.bPressed				:= tyInternal.fbTouchFilter.bPressedOut;
		tyInternal.fbTouchGetTap.udiX					:= tyInternal.fbTouchFilter.udiXOut;
		tyInternal.fbTouchGetTap.udiY					:= tyInternal.fbTouchFilter.udiYOut;
		tyInternal.fbTouchGetTap;

		fUIInRtStatOff(ADR(p_uiSliderStatus));

		IF tyInternal.fbTouchFilter.bPressedOut = TRUE THEN
			tyInternal.fbSliderOffTm(IN := FALSE);
			tyInternal.fbSingleTapChkDlyTm(IN := FALSE);

			IF uiSlideScale < 1 THEN
				uiSlideScale	:= 1;
			END_IF

			tyInternal.iTablePos	:= tyInternal.iTablePosTemp - DINT_TO_INT(tyInternal.fbTouchGetSlideDist.diYDist) / UINT_TO_INT(uiSlideScale);

			IF tyInternal.iTablePos > (iTotalData - iTotalRow + 1) THEN
				IF (iTotalData - iTotalRow + 1) < 1 THEN
					tyInternal.iTablePos	:= 1;
				ELSE
					tyInternal.iTablePos	:= iTotalData - iTotalRow + 1;
				END_IF

			ELSIF tyInternal.iTablePos < 1 THEN
				tyInternal.iTablePos	:= 1;

			END_IF

			p_uiTablePos	:= INT_TO_UINT(tyInternal.iTablePos);
			p_iSliderPos	:= UINT_TO_INT(p_uiTablePos);

		ELSE
			tyInternal.iTablePosTemp	:= tyInternal.iTablePos;

			tyInternal.fbSingleTapChkDlyTm(IN := TRUE);

			IF tyInternal.fbSingleTapChkDlyTm.Q = TRUE THEN
				FOR tyInternal.i := 1 TO 15 DO
					pa_tyUIHotspot[tyInternal.i].bRtCompl	:= FALSE;
				END_FOR

				p_bTableActive	:= FALSE;

			ELSE
				FOR tyInternal.i := 1 TO 15 DO
					IF pa_tyUIHotspot[tyInternal.i].bValue = TRUE THEN
						IF tyInternal.fbTouchGetTap.bSingleTap = TRUE THEN
							p_uiSelectedRow	:= tyInternal.i;
						END_IF

						pa_tyUIHotspot[tyInternal.i].bValue	:= FALSE;

					END_IF

				END_FOR

			END_IF

		END_IF

	ELSIF p_uiSliderStatus.0 = FALSE THEN
		tyInternal.fbSliderOffTm(IN := TRUE);

		IF tyInternal.fbSliderOffTm.Q = TRUE THEN
			fUIInRtStatHide(ADR(p_uiSliderStatus));
			tyInternal.fbSliderOffTm(IN := FALSE);

		END_IF

	END_IF

	tyInternal.fbSelectedRowMnlRise(CLK := bSelectedRowMnl);
	IF tyInternal.fbSelectedRowMnlRise.Q THEN
		p_uiSelectedRow	:= uiSelectedRowMnl;
	END_IF

	tyInternal.fbTablePosUpRise(CLK := bTablePosPlus);
	IF tyInternal.fbTablePosUpRise.Q THEN
		p_uiTablePos				:= p_uiTablePos + 1;
		p_iSliderPos				:= p_iSliderPos + 1;
		tyInternal.iTablePos		:= tyInternal.iTablePos + 1;
		tyInternal.iTablePosTemp	:= tyInternal.iTablePosTemp + 1;

	END_IF

	tyInternal.fbTablePosDownRise(CLK := bTablePosMinus);
	IF tyInternal.fbTablePosDownRise.Q THEN
		p_uiTablePos				:= p_uiTablePos - 1;
		p_iSliderPos				:= p_iSliderPos - 1;
		tyInternal.iTablePos		:= tyInternal.iTablePos - 1;
		tyInternal.iTablePosTemp	:= tyInternal.iTablePosTemp - 1;

	END_IF

END_FUNCTION_BLOCK
```

#### fbTouchFilter.st
```iecst
(* Filter Touch Action *)
FUNCTION_BLOCK fbTouchFilter

	IF bPressedIn = TRUE THEN
		tyInternal.udiXOld	:= udiXIn;
		tyInternal.udiYOld	:= udiYIn;

		bPressedOut	:= TRUE;
		udiXOut		:= udiXIn;
		udiYOut		:= udiYIn;

	ELSIF (bPressedIn = FALSE) AND (tyInternal.udiXOld <> udiXIn OR tyInternal.udiYOld <> udiYIn) AND (tyInternal.udiXOld = 0 AND tyInternal.udiYOld = 0) THEN
		tyInternal.udiXOld	:= udiXIn;
		tyInternal.udiYOld	:= udiYIn;

		bPressedOut	:= FALSE;
		udiXOut		:= udiXIn;
		udiYOut		:= udiYIn;

	ELSIF (bPressedIn = FALSE) AND (tyInternal.udiXOld <> udiXIn OR tyInternal.udiYOld <> udiYIn) THEN
		tyInternal.udiXOld	:= udiXIn;
		tyInternal.udiYOld	:= udiYIn;

		bPressedOut	:= TRUE;
		udiXOut		:= udiXIn;
		udiYOut		:= udiYIn;

	ELSE
		bPressedOut	:= FALSE;

	END_IF

END_FUNCTION_BLOCK
```

### Library Logical/NtLibraries/NtGeneral (IEC, version 5.00.1) - 5.00.1 - Add tyAlmTxt
5.00.0 - New Library Design. (20181211)

#### NtGeneral.fun - Exported functions and function blocks
```iecst
FUNCTION_BLOCK fbSenFltr (*Filter Sensor With Time*) (*$GROUP=Nutek,$CAT=User,$GROUPICON=Icon_Nutek.png,$CATICON=User.png*)
	VAR_INPUT
		bSigIn : {REDUND_UNREPLICABLE} BOOL; (*Sensor Input*)
		tSigOnFltrTm : {REDUND_UNREPLICABLE} TIME; (*Sensor Signal On Filter Time*)
		tSigOffFltrTm : {REDUND_UNREPLICABLE} TIME; (*Sensor Signal Off Filter Time*)
	END_VAR
	VAR_OUTPUT
		bSigOut : BOOL; (*Output - Sensor Output*)
	END_VAR
	VAR
		tyInternal : {REDUND_UNREPLICABLE} tySenFltrInternal; (*Local Variables*)
	END_VAR
END_FUNCTION_BLOCK

FUNCTION fValidCharStringInChkr : BOOL (*Valid Character For String Input Checker*) (*$GROUP=Nutek,$CAT=User,$GROUPICON=Icon_Nutek.png,$CATICON=User.png*)
	VAR_INPUT
		p_sMismatchChar : REFERENCE TO STRING[1]; (*Output - Mismatch Character*)
		sInChk : STRING[255]; (*String Input To Be Checked*)
		sValidMember : STRING[128]; (*Valid String Members For Checking*)
	END_VAR
	VAR
		tyInternal : tyValidCharChkrInternal; (*Local Variables*)
	END_VAR
END_FUNCTION

FUNCTION fInvalidCharStringInChkr : BOOL (*Invalid Character For String Input Checker*) (*$GROUP=Nutek,$CAT=User,$GROUPICON=Icon_Nutek.png,$CATICON=User.png*)
	VAR_INPUT
		p_sInvalidChar : REFERENCE TO STRING[1]; (*Output - Invalid Character*)
		sInChk : STRING[255]; (*String Input To Be Checked*)
		sInvalidMember : STRING[128]; (*Invalid String Members For Checking*)
	END_VAR
	VAR
		tyInternal : tyInvalidCharChkrInternal; (*Local Variables*)
	END_VAR
END_FUNCTION

FUNCTION fCheckDuplicate : USINT (*Check Input Value Duplicate*) (*$GROUP=Nutek,$CAT=User,$GROUPICON=Icon_Nutek.png,$CATICON=User.png*)
	VAR_INPUT
		a_usiValue : ARRAY[1..100] OF USINT; (*Value to Check*)
		a_bChkValue : ARRAY[1..100] OF BOOL; (*True = Check Value, False = No Need Check*)
	END_VAR
	VAR
		tyInternal : tyCheckDuplicateInternal; (*Local Variables*)
	END_VAR
END_FUNCTION

FUNCTION fCheckExist : USINT (*Check Exist Of Value*) (*$GROUP=Nutek,$CAT=User,$GROUPICON=Icon_Nutek.png,$CATICON=User.png*)
	VAR_INPUT
		a_usiValue : ARRAY[1..50] OF USINT; (*Value to Check*)
		a_bChkValue : ARRAY[1..50] OF BOOL; (*True = Check Value, False = No Need Check*)
	END_VAR
	VAR
		tyInternal : tyCheckExistInternal; (*Local Variables*)
	END_VAR
END_FUNCTION

FUNCTION fStringSearch : UDINT (*String Search*) (*$GROUP=Nutek,$CAT=User,$GROUPICON=Icon_Nutek.png,$CATICON=User.png*)
	VAR_INPUT
		p_StringChk : UDINT; (*Address Of String Input To Be Checked*)
		udiStringChkSize : UDINT; (*Size of String Input To Be Checked*)
		sSearch : STRING[255]; (*String Search*)
	END_VAR
	VAR
		tyInternal : tyStringSearchInternal; (*Local Variables*)
	END_VAR
END_FUNCTION

FUNCTION fIPValid : BOOL (*Check IP Address Validation*) (*$GROUP=Nutek,$CAT=User,$GROUPICON=Icon_Nutek.png,$CATICON=User.png*)
	VAR_INPUT
		sIPAdd : STRING[15] := ''; (*IP Address*)
		pa_iIPPart : REFERENCE TO ARRAY[1..4] OF INT; (*IP Address Part in Integer*)
	END_VAR
	VAR
		tyInternal : tyIPValidInternal;
	END_VAR
END_FUNCTION

FUNCTION fConvertUINTToHex : BOOL (*Convert UINT To Hex*)
	VAR_INPUT
		p_sHexOut : REFERENCE TO STRING[4]; (*Output - Hex*)
		uiDecimalIn : UINT; (*Decimal Input*)
	END_VAR
	VAR
		uiTemp1 : UINT;
		uiTemp2 : UINT;
	END_VAR
END_FUNCTION

FUNCTION fConvertUSINTToHex : BOOL (*Convert USINT To Hex*)
	VAR_INPUT
		p_sHexOut : REFERENCE TO STRING[2]; (*Output - Hex*)
		usiDecimalIn : USINT; (*Decimal Input*)
	END_VAR
	VAR
		usiTemp1 : USINT;
		usiTemp2 : USINT;
	END_VAR
END_FUNCTION

FUNCTION fConvertToLower_254 : BOOL (*Convert Input STRING to Lower Case*)
	VAR_INPUT
		p_sOutput : REFERENCE TO STRING[254]; (*Output - String*)
		sInput : STRING[254]; (*Input String*)
	END_VAR
	VAR
		udi : UDINT;
		si : SINT;
	END_VAR
END_FUNCTION
```

#### Types.typ - Exported data types
```iecst
(*Library Status*)

TYPE
	eFBStatus :
		( (*Function Block Status*)
		Idle, (*Library In Idle Status*)
		Done, (*Library In Done Status*)
		Busy, (*Library In Busy Status*)
		Error (*Library In Error Status*)
		);
END_TYPE

(**)
(*Alarm*)

TYPE
	tyAlmTxt : 	STRUCT
		sAlmText : STRING[200]; (*Alarm Text*)
		sRcyText : STRING[200]; (*Recovery Text*)
	END_STRUCT;
	tyAlmDat : 	STRUCT
		udiCode : UDINT; (*Alarm Code*)
		eSeverity : eAlmSeverity; (*Alarm Severity*)
		sProgNm : STRING[15]; (*Program Title Name*)
		sAlmMsg : STRING[200]; (*Alarm Message*)
		sRcyMsg : STRING[200]; (*Recovery Message*)
		udiRunTime : UDINT; (*Run Time*)
		udiModuleNum : UDINT;
		bAlm : BOOL;
		bWarning : BOOL;
	END_STRUCT;
	eAlmSeverity :
		(
		AlmSeverityNA, (*Error*)
		AlmSeverityError, (*Error*)
		AlmSeverityWarning, (*Warning*)
		AlmSeverityInfo (*Information*)
		);
	tyAlmInputProps : 	STRUCT
		uiModuleOrder : UINT;
	END_STRUCT;
END_TYPE

(*Others*)

TYPE
	tyValidCharChkrInternal : {REDUND_UNREPLICABLE} 	STRUCT  (*Local Variables*)
		sValidChar : {REDUND_UNREPLICABLE} STRING[1]; (*Valid Characters For Checking*)
		sCharChk : {REDUND_UNREPLICABLE} STRING[1]; (*Character On Checking*)
		i : {REDUND_UNREPLICABLE} INT;
		j : {REDUND_UNREPLICABLE} INT;
	END_STRUCT;
	tyInvalidCharChkrInternal : {REDUND_UNREPLICABLE} 	STRUCT  (*Local Variables*)
		sInvalidChar : {REDUND_UNREPLICABLE} STRING[1]; (*Invalid Characters For Checking*)
		sCharChk : {REDUND_UNREPLICABLE} STRING[1]; (*Character On Checking*)
		i : {REDUND_UNREPLICABLE} INT;
		j : {REDUND_UNREPLICABLE} INT;
	END_STRUCT;
	tyCheckDuplicateInternal : {REDUND_UNREPLICABLE} 	STRUCT  (*Local Variables*)
		i : {REDUND_UNREPLICABLE} USINT;
		j : {REDUND_UNREPLICABLE} USINT;
		usiCnt : {REDUND_UNREPLICABLE} USINT; (*Counter*)
	END_STRUCT;
	tyStringSearchInternal : {REDUND_UNREPLICABLE} 	STRUCT  (*Local Variables*)
		i : {REDUND_UNREPLICABLE} UDINT;
		usiZero : {REDUND_UNREPLICABLE} USINT; (*Counter*)
	END_STRUCT;
	tyCheckExistInternal : {REDUND_UNREPLICABLE} 	STRUCT  (*Local Variables*)
		i : {REDUND_UNREPLICABLE} USINT;
		j : {REDUND_UNREPLICABLE} USINT;
		usiCnt : {REDUND_UNREPLICABLE} USINT; (*Counter*)
	END_STRUCT;
	tySenFltrInternal : {REDUND_UNREPLICABLE} 	STRUCT  (*Local Variables*)
		fbSigFltrTm : {REDUND_UNREPLICABLE} TON; (*Signal Filter Time*)
	END_STRUCT;
	tyIPValidInternal : 	STRUCT  (*Local Variables*)
		i : INT;
		iCnt : INT; (*Counter*)
		a_iDotPos : ARRAY[1..3]OF INT; (*IP Address Dot Position*)
		a_sIPPart : ARRAY[1..4]OF STRING[3]; (*IP Address Part in String*)
		a_iIPPart : ARRAY[1..4]OF INT; (*IP Address Part in Integer*)
		sMismatchChar : STRING[1]; (*Mismatch Character*)
	END_STRUCT;
END_TYPE
```

#### fbSenFltr.st
```iecst
(* Filter Sensor With Time *)
FUNCTION_BLOCK fbSenFltr

	IF bSigIn = TRUE AND bSigOut = FALSE THEN
		tyInternal.fbSigFltrTm(IN := TRUE , PT := tSigOnFltrTm);
		IF tyInternal.fbSigFltrTm.Q = TRUE THEN
			bSigOut	:= TRUE;
		END_IF

	ELSIF bSigIn = FALSE AND bSigOut = TRUE THEN
		tyInternal.fbSigFltrTm(IN := TRUE , PT := tSigOffFltrTm);
		IF tyInternal.fbSigFltrTm.Q = TRUE THEN
			bSigOut	:= FALSE;
		END_IF

	ELSE
		tyInternal.fbSigFltrTm(IN := FALSE);

	END_IF

END_FUNCTION_BLOCK
```

#### fValidCharStringInChkr.st
```iecst
(* Valid Character For String Input Checker *)
FUNCTION fValidCharStringInChkr

	// Valid character for string input checker
	// Valid characters match for string input: bValid = TRUE
	// Mismatch character can be observed on p_sMismatchChar
	//--------------------------------------------------------------------------------
	fValidCharStringInChkr	:= TRUE;
	p_sMismatchChar 		:= '';

	FOR tyInternal.i := 0 TO LEN(sInChk) - 1 DO
		memmove(ADR(tyInternal.sCharChk) , ADR(sInChk) + INT_TO_UDINT(tyInternal.i) , 1);

		fValidCharStringInChkr	:= FALSE;

		FOR tyInternal.j := 0 TO LEN(sValidMember) - 1 DO
			memmove(ADR(tyInternal.sValidChar) , ADR(sValidMember) + INT_TO_UDINT(tyInternal.j) , 1);

			IF memcmp(ADR(tyInternal.sCharChk) , ADR(tyInternal.sValidChar) , 1) = 0 THEN
				fValidCharStringInChkr := TRUE;
				EXIT;
			END_IF
		END_FOR

		IF fValidCharStringInChkr = FALSE THEN
			p_sMismatchChar	:= tyInternal.sCharChk;
			EXIT;
		END_IF
	END_FOR

END_FUNCTION
```

#### fInvalidCharStringInChkr.st
```iecst
(* Invalid Character For String Input Checker *)
FUNCTION fInvalidCharStringInChkr

	// Invalid character for string input checker
	// Invalid characters match for string input: bValid = TRUE
	// Match Invalid character can be observed on p_sInvalidChar
	//--------------------------------------------------------------------------------

	p_sInvalidChar := '';

	FOR tyInternal.i := 0 TO LEN(sInChk) - 1 DO
		memmove(ADR(tyInternal.sCharChk) , ADR(sInChk) + tyInternal.i , 1);
		fInvalidCharStringInChkr := FALSE;

		FOR tyInternal.j := 0 TO LEN(sInvalidMember) - 1 DO
			memmove(ADR(tyInternal.sInvalidChar) , ADR(sInvalidMember) + tyInternal.j , 1);

			IF memcmp(ADR(tyInternal.sCharChk) , ADR(tyInternal.sInvalidChar) , 1) = 0 THEN
				fInvalidCharStringInChkr := TRUE;
				EXIT;
			END_IF
		END_FOR

		IF fInvalidCharStringInChkr THEN
			p_sInvalidChar := tyInternal.sCharChk;
			EXIT;
		END_IF
	END_FOR

END_FUNCTION
```

#### fCheckDuplicate.st
```iecst
(* Check Input Duplicate *)
FUNCTION fCheckDuplicate

	fCheckDuplicate	:= 0;

	FOR tyInternal.i := 1 TO 100 DO
		IF a_bChkValue[tyInternal.i] = TRUE THEN

			tyInternal.usiCnt	:= 0;

			FOR tyInternal.j := 1 TO 100 DO
				IF a_usiValue[tyInternal.j] = tyInternal.i THEN
					tyInternal.usiCnt	:= tyInternal.usiCnt + 1;

					IF tyInternal.usiCnt > 1 THEN
						fCheckDuplicate	:= tyInternal.i;
						EXIT;
					END_IF

				END_IF

			END_FOR

			IF fCheckDuplicate <> 0 THEN
				EXIT;
			END_IF

		END_IF

	END_FOR

END_FUNCTION
```

#### fCheckExist.st
```iecst
(* Check Exist Of Value *)
FUNCTION fCheckExist

	fCheckExist	:= 0;

	FOR tyInternal.i := 1 TO 50 DO
		IF a_bChkValue[tyInternal.i] = TRUE THEN

			FOR tyInternal.j := 1 TO 50 DO
				IF a_usiValue[tyInternal.j] = tyInternal.i THEN
					EXIT;
				END_IF
			END_FOR

			IF tyInternal.j = 51 THEN
				fCheckExist	:= tyInternal.i;
				EXIT;
			END_IF

		END_IF

	END_FOR

END_FUNCTION
```

#### fStringSearch.st
```iecst
(* String Search *)
FUNCTION fStringSearch

	fStringSearch	:= 0;

	IF udiStringChkSize < INT_TO_UDINT(LEN(sSearch)) THEN
		;
	ELSE
		FOR tyInternal.i := p_StringChk TO (p_StringChk + udiStringChkSize - LEN(sSearch) + 1) DO
			IF memcmp(ADR(sSearch) , tyInternal.i , LEN(sSearch)) = 0 THEN
				fStringSearch	:= tyInternal.i - p_StringChk + 1;
				EXIT;
			ELSIF memcmp(tyInternal.i , ADR(tyInternal.usiZero) , 1) = 0 THEN
				EXIT;
			END_IF
		END_FOR
	END_IF

END_FUNCTION
```

#### fIPValid.st
```iecst
(* Check IP Address Validation *)
FUNCTION fIPValid

	fIPValid	:= FALSE;
	memset(ADR(pa_iIPPart) , 0 , SIZEOF(pa_iIPPart));

	IF fValidCharStringInChkr(ADR(tyInternal.sMismatchChar) , sIPAdd , '1234567890.') = TRUE THEN
		IF LEN(sIPAdd) >= 7 AND LEN(sIPAdd) <= 15 THEN
			memset(ADR(tyInternal.a_iDotPos) , 0 , SIZEOF(tyInternal.a_iDotPos));
			memset(ADR(tyInternal.a_sIPPart) , 0 , SIZEOF(tyInternal.a_sIPPart));
			memset(ADR(pa_iIPPart) , 0 , SIZEOF(pa_iIPPart));
			tyInternal.iCnt	:= 0;

			FOR tyInternal.i := 0 TO LEN(sIPAdd) -1 DO
				IF memcmp(ADR(sIPAdd) + tyInternal.i , ADR('.') , 1) = 0 THEN
					tyInternal.iCnt	:= tyInternal.iCnt + 1;
					IF tyInternal.iCnt < 4 THEN
						tyInternal.a_iDotPos[tyInternal.iCnt]	:= tyInternal.i + 1;
					ELSE
						EXIT;
					END_IF
				END_IF
			END_FOR

			IF tyInternal.iCnt = 3 THEN
				memcpy(ADR(tyInternal.a_sIPPart[1]) , ADR(sIPAdd) , tyInternal.a_iDotPos[1] - 1);
				memcpy(ADR(tyInternal.a_sIPPart[2]) , ADR(sIPAdd) + tyInternal.a_iDotPos[1] , tyInternal.a_iDotPos[2] - tyInternal.a_iDotPos[1] - 1);
				memcpy(ADR(tyInternal.a_sIPPart[3]) , ADR(sIPAdd) + tyInternal.a_iDotPos[2] , tyInternal.a_iDotPos[3] - tyInternal.a_iDotPos[2] - 1);
				memcpy(ADR(tyInternal.a_sIPPart[4]) , ADR(sIPAdd) + tyInternal.a_iDotPos[3] , LEN(sIPAdd) - tyInternal.a_iDotPos[3]);

				IF tyInternal.a_sIPPart[1] <> '' AND tyInternal.a_sIPPart[2] <> '' AND tyInternal.a_sIPPart[3] <> '' AND tyInternal.a_sIPPart[4] <> '' THEN
					FOR tyInternal.i := 1 TO 4 DO
						pa_iIPPart[tyInternal.i]	:= STRING_TO_INT(tyInternal.a_sIPPart[tyInternal.i]);
					END_FOR

					IF pa_iIPPart[1] >= 1 AND pa_iIPPart[1] <= 255 AND pa_iIPPart[2] >= 0 AND pa_iIPPart[2] <= 255 AND pa_iIPPart[3] >= 0 AND pa_iIPPart[3] <= 255 AND pa_iIPPart[4] >= 0 AND pa_iIPPart[4] <= 255 THEN
						fIPValid	:= TRUE;
					END_IF
				END_IF
			END_IF
		END_IF
	END_IF

END_FUNCTION
```

#### fConvertUINTToHex.st
```iecst
(* Convert UINT To Hex *)
FUNCTION fConvertUINTToHex

	fConvertUINTToHex	:= TRUE;

	uiTemp1		:= uiDecimalIn;
	p_sHexOut	:= '';

	WHILE uiTemp1 <> 0 DO
		uiTemp2	:= uiTemp1 MOD 16;
		uiTemp1	:= uiTemp1 / 16;

		CASE uiTemp2 OF
			0:		p_sHexOut	:= CONCAT('0' , p_sHexOut);
			1:		p_sHexOut	:= CONCAT('1' , p_sHexOut);
			2:		p_sHexOut	:= CONCAT('2' , p_sHexOut);
			3:		p_sHexOut	:= CONCAT('3' , p_sHexOut);
			4:		p_sHexOut	:= CONCAT('4' , p_sHexOut);
			5:		p_sHexOut	:= CONCAT('5' , p_sHexOut);
			6:		p_sHexOut	:= CONCAT('6' , p_sHexOut);
			7:		p_sHexOut	:= CONCAT('7' , p_sHexOut);
			8:		p_sHexOut	:= CONCAT('8' , p_sHexOut);
			9:		p_sHexOut	:= CONCAT('9' , p_sHexOut);
			10:		p_sHexOut	:= CONCAT('A' , p_sHexOut);
			11:		p_sHexOut	:= CONCAT('B' , p_sHexOut);
			12:		p_sHexOut	:= CONCAT('C' , p_sHexOut);
			13:		p_sHexOut	:= CONCAT('D' , p_sHexOut);
			14:		p_sHexOut	:= CONCAT('E' , p_sHexOut);
			ELSE	p_sHexOut	:= CONCAT('F' , p_sHexOut);
		END_CASE

	END_WHILE

	IF LEN(p_sHexOut) = 0 THEN
		p_sHexOut	:= CONCAT('0000' , p_sHexOut);
	ELSIF LEN(p_sHexOut) = 1 THEN
		p_sHexOut	:= CONCAT('000' , p_sHexOut);
	ELSIF LEN(p_sHexOut) = 2 THEN
		p_sHexOut	:= CONCAT('00' , p_sHexOut);
	ELSIF LEN(p_sHexOut) = 3 THEN
		p_sHexOut	:= CONCAT('0' , p_sHexOut);
	END_IF

END_FUNCTION
```

#### fConvertUSINTToHex.st
```iecst
(* Convert USINT To Hex *)
FUNCTION fConvertUSINTToHex

	fConvertUSINTToHex	:= TRUE;

	usiTemp1	:= usiDecimalIn;
	p_sHexOut	:= '';

	WHILE usiTemp1 <> 0 DO
		usiTemp2	:= usiTemp1 MOD 16;
		usiTemp1	:= usiTemp1 / 16;

		CASE usiTemp2 OF
			0:		p_sHexOut	:= CONCAT('0' , p_sHexOut);
			1:		p_sHexOut	:= CONCAT('1' , p_sHexOut);
			2:		p_sHexOut	:= CONCAT('2' , p_sHexOut);
			3:		p_sHexOut	:= CONCAT('3' , p_sHexOut);
			4:		p_sHexOut	:= CONCAT('4' , p_sHexOut);
			5:		p_sHexOut	:= CONCAT('5' , p_sHexOut);
			6:		p_sHexOut	:= CONCAT('6' , p_sHexOut);
			7:		p_sHexOut	:= CONCAT('7' , p_sHexOut);
			8:		p_sHexOut	:= CONCAT('8' , p_sHexOut);
			9:		p_sHexOut	:= CONCAT('9' , p_sHexOut);
			10:		p_sHexOut	:= CONCAT('A' , p_sHexOut);
			11:		p_sHexOut	:= CONCAT('B' , p_sHexOut);
			12:		p_sHexOut	:= CONCAT('C' , p_sHexOut);
			13:		p_sHexOut	:= CONCAT('D' , p_sHexOut);
			14:		p_sHexOut	:= CONCAT('E' , p_sHexOut);
			ELSE	p_sHexOut	:= CONCAT('F' , p_sHexOut);
		END_CASE

	END_WHILE

	IF LEN(p_sHexOut) = 0 THEN
		p_sHexOut	:= CONCAT('00' , p_sHexOut);
	ELSIF LEN(p_sHexOut) = 1 THEN
		p_sHexOut	:= CONCAT('0' , p_sHexOut);
	END_IF

END_FUNCTION
```

#### fConvertToLower_254.st
```iecst
(* Convert Input STRING to Lower Case *)
FUNCTION fConvertToLower_254

	fConvertToLower_254	:= TRUE;

	p_sOutput	:= sInput;

	FOR udi := 0 TO LEN(sInput) DO

		memcpy(ADR(si) , ADR(sInput) + udi , 1);

		IF si >= 65 AND si <= 90 THEN
			si	:= si + 32;
			memcpy(ADR(p_sOutput) + udi , ADR(si) , 1);
		ELSIF si = 0 THEN
			EXIT;
		END_IF

	END_FOR

END_FUNCTION
```

### Library Logical/NtLibraries/NtHermes (IEC, version 5.00.4) - 5.00.4 - Hermes v1.3
5.00.3 - Debug of fHermesGetTimeStamp.(20191029)
5.00.2 - Add for Remote Configuration. (20190504)
5.00.1 - Debug fHermesIllegalMsgBrdAvlDS. (20190425)
5.00.0 - New Library Design. (20181221)
Depends on: NtGeneral
